// §6.9/§3.10(a') — overlay the pending stall after the common mirror refresh.
METHOD PROTECTED _M_PublishStatus
SUPER^._M_PublishStatus();
// §8.11.4(f)/§8.11.3 — one declaration, two views. Derived AFTER dispatch so the
// wait class reflects the step record this scan just set, not the previous one.
// §3.13 — live row state for the flow chart: how long the active step has run,
// and whether it outran its declared guard (the same watchdog §6.9 stalls on).
IF _exec = E_ExecState.BUSY THEN
    CurrentStepElapsed := DWORD_TO_TIME(TIME_TO_DWORD(TIME()) - _stepSinceMs);
ELSE
    CurrentStepElapsed := T#0S;
END_IF
CurrentStepTimedOut := _tStall.Q;
Starved := (_exec = E_ExecState.BUSY) AND (CurrentStep.TimeClass = E_TimeClass.WAIT_UPSTREAM);
Blocked := (_exec = E_ExecState.BUSY) AND (CurrentStep.TimeClass = E_TimeClass.WAIT_DOWNSTREAM);
// §8.11.3 — classify into the fixed machine-state set (priority: fault first,
// then planned states, then line attribution, then producing/idle).
IF (_exec = E_ExecState.ERROR) OR AlarmLog.Blocking THEN
    MachineState := E_MachineState.DOWN;
ELSIF _mode = E_Mode.CHANGEOVER THEN
    MachineState := E_MachineState.CHANGEOVER;
ELSIF Blocked THEN
    MachineState := E_MachineState.BLOCKED;
ELSIF Starved THEN
    MachineState := E_MachineState.STARVED;
ELSIF _exec = E_ExecState.BUSY THEN
    MachineState := E_MachineState.PRODUCING;
ELSIF _stopReq OR (_exec = E_ExecState.ABORTED) THEN
    MachineState := E_MachineState.STOPPED;
ELSE
    MachineState := E_MachineState.IDLE;
END_IF
Status.ControlDomainId := ControlDomain.Id;
Domain := ControlDomain;
Safety := ControlDomain.Safety;             // read-only HMI mirror; ownership stays in domain
ControlPower := ControlDomain.ControlPower;
IF (_exec <> E_ExecState.ERROR) AND (Pending.ReasonCode <> E_Reason.NONE) THEN
    Status.Diagnostic := Pending;
END_IF
END_METHOD

// §6.9(a) — fixed ring, newest at HistoryHead; never allocates
METHOD PROTECTED _M_PushHistory
VAR_INPUT
    D : ST_Diagnostic;
END_VAR
HistoryHead := (HistoryHead MOD PL_Fraktal.MAX_DIAG_RING) + 1;
History[HistoryHead] := D;
END_METHOD

// §8.11.4(d)/§8.12 — a Low-severity maintenance event: informs planning, does not
// stop the cycle. Instant come+gone ring entry (the trend data lives in Profiler).
METHOD PROTECTED _M_RaiseMaintenance
VAR_INPUT
    Reason : E_Reason;
    Text : STRING(255);
END_VAR
VAR
    slot : INT;
END_VAR
slot := AlarmLog.Raise(Reason := Reason, Text := Text, Source := _name,
    Severity := E_Severity.LOW, Category := E_Category.SYSTEM,
    ResetClass := E_ResetClass.AUTO_RESET);
IF slot > 0 THEN
    AlarmLog.Gone(Slot := slot);
END_IF
END_METHOD

// §3.8b — route a published editable field to the module that registered it.
// WriteConfig already owns access and root-path checks; the recursive walk finds
// the owner by Scope, and that module rechecks revision, type, range, domain and
// its own invariants before storing. A type whose values are declared through
// M_RegisterConfig* therefore needs no override at all, which is the point: a new
// module type costs no routing code (§1.1 O1). Framework-owned keys never reach
// here — _M_WriteBaseConfig answers those first. An override that adds
// hand-written routing shall call SUPER^ first and keep its own answer only when
// the base declines.
METHOD PROTECTED _M_RouteConfigWrite : BOOL
VAR_INPUT
    TargetPath : STRING(255);
    WriteKey   : STRING(160);
    Revision   : UDINT;
    TextValue  : STRING(255);
END_VAR
// RequiresReady is a question about THIS root's state, which the owning child
// cannot see from where it sits, so the root answers it on the way down.
_M_RouteConfigWrite := M_ApplyConfigWrite(Scope := TargetPath,
    WriteKey := WriteKey, Revision := Revision, TextValue := TextValue,
    // Another model's record is not what the machine is running on.
    RootReady := (_exec = E_ExecState.READY) OR (_pModelView <> 0));
END_METHOD

// Framework-owned typed handlers. Stable keys are independent of browse paths;
// capability revision 1 accepts exact enum ordinals and only while READY.
//
// Commit := FALSE validates and stores nothing — the staging pass of a §3.8b set
// load. The root's own ModePolicy keys are published as STATION_CFG
// capabilities, so they are in every station set and have to stage through the
// same validator that writes them, for the same reason every module's do.
METHOD PRIVATE _M_WriteBaseConfig : BOOL
VAR_INPUT
    TargetPath : STRING(255);
    WriteKey   : STRING(160);
    Revision   : UDINT;
    TextValue  : STRING(255);
    Commit     : BOOL;
END_VAR
VAR
    i      : INT;
    key    : STRING(160);
    shield : E_ModeSwitchShield;
    style  : E_ModeSwitchStyle;
END_VAR
_M_WriteBaseConfig := FALSE;
IF (TargetPath <> Status.Name) OR (Revision <> 1) OR (_exec <> E_ExecState.READY) THEN
    RETURN;
END_IF
FOR i := 0 TO PL_Fraktal.MODE_COUNT - 1 DO
    key := CONCAT('unit.modePolicy.', CONCAT(TO_STRING(i), '.shield'));
    IF WriteKey = key THEN
        IF TextValue = '0' THEN
            shield := E_ModeSwitchShield.INTERRUPTIBLE;
        ELSIF TextValue = '1' THEN
            shield := E_ModeSwitchShield.CONFIRM;
        ELSIF TextValue = '2' THEN
            shield := E_ModeSwitchShield.BLOCKED_WHILE_RUNNING;
        ELSE
            RETURN;
        END_IF
        IF Commit THEN
            ModePolicy[i].Shield := shield;
            _modePolicyStored[i].Shield := shield;
        END_IF
        _M_WriteBaseConfig := TRUE;
        RETURN;
    END_IF
    key := CONCAT('unit.modePolicy.', CONCAT(TO_STRING(i), '.style'));
    IF WriteKey = key THEN
        IF TextValue = '0' THEN
            style := E_ModeSwitchStyle.GRACEFUL;
        ELSIF TextValue = '1' THEN
            style := E_ModeSwitchStyle.IMMEDIATE;
        ELSE
            RETURN;
        END_IF
        IF Commit THEN
            ModePolicy[i].Style := style;
            _modePolicyStored[i].Style := style;
        END_IF
        _M_WriteBaseConfig := TRUE;
        RETURN;
    END_IF
END_FOR
END_METHOD

// Application override resolves ChannelPath in THIS root's approved I/O catalog,
// refuses input/safety/unmapped channels, applies its channel-specific §7.6 permit,
// and routes only an approved mapped output. ForceChannel already owns MANUAL,
// stopped/READY, access and audit. Base fails closed.
METHOD PROTECTED _M_RouteForceChannel : BOOL
VAR_INPUT
    ChannelPath : STRING(255);
    Force       : BOOL;
    BoolText    : STRING(255);
    AnalogText  : STRING(160);
END_VAR
_M_RouteForceChannel := FALSE;
END_METHOD

// §7.6.1 — route a manual command to the module that owns TargetPath, through
// the SAME registered-child walk that already carries configuration writes.
//
// This used to return FALSE and leave every Unit to hand-write its own routing
// chain. That is a call a project must remember for correctness (§1.1 O1), and
// it failed exactly as O1 predicts: the press registered eight children and
// routed three, so five modules published manual commands the HMI rendered and
// the Unit silently refused. A registered child is now commandable BECAUSE it
// is registered.
//
// An override still wins, so a Unit with genuinely special routing keeps it;
// it should call SUPER^ first and keep its own answer only when the base
// declines.
METHOD PROTECTED _M_RouteManual : BOOL
VAR_INPUT
    TargetPath : STRING(255);
    Value : DINT;
END_VAR
_M_RouteManual := M_ApplyManual(Scope := TargetPath, Value := Value);
END_METHOD

// §3.13 — keep the published flow chart in step with the chain.
// Called only from _M_SetStep, so every step of every chain lands here exactly
// once per visit and a chain author writes nothing (§1.1 O1). Rows are matched by
// StepNo, appended on first sight and bounded: an overflowing chain publishes the
// first MAX_SEQUENCE_STEPS rows rather than dropping the chart.
METHOD PROTECTED _M_RecordSequenceStep
VAR_INPUT
    StepNo        : INT;
    StepName      : STRING(120);
    Awaits        : I_Module;
    AwaitingLabel : STRING(120);
    TimeClass     : E_TimeClass;
    ExpectedTime  : TIME;
    Branch        : INT;           // §6.12 concurrent leg, 0 = the chain's main line
END_VAR
VAR
    i    : INT;
    hit  : INT;
    path : STRING(255);
END_VAR
hit := 0;
FOR i := 1 TO SequenceStepCount DO
    IF SequenceStepDef[i].StepNo = StepNo THEN
        hit := i;
        EXIT;
    END_IF
END_FOR
IF hit = 0 THEN
    IF SequenceStepCount >= PL_Fraktal.MAX_SEQUENCE_STEPS THEN
        RETURN;                        // bounded: publish what fits, never overrun
    END_IF
    SequenceStepCount := SequenceStepCount + 1;
    hit := SequenceStepCount;
    // §3.10.2 — the static half of this row (StepNo, StepName, the awaited path)
    // is served through the manifest, NOT cyclically, and the HMI refetches only
    // when ConfigRev changes. Rows are discovered by visit, so a chart that grows
    // after the HMI's fetch would render every new row with StepNo 0 and no text.
    // Only the append marks it: a re-visit rewrites identical values.
    //
    // MARKED, not bumped: the revision is raised once the chart stops growing
    // (_M_ChartRevCyclic). Invalidating the whole manifest per discovered row
    // made entering a 15-step mode cost fifteen full refetches.
    _chartDirty := TRUE;
    _chartTouchedMs := TIME_TO_DWORD(TIME());
END_IF
// The drill-down target is the module the step DECLARES it commands. Reading it
// here is what makes the link unambiguous: no IF/CASE chose it (§3.13).
path := '';
IF Awaits <> 0 THEN
    path := Awaits.Name;
END_IF
// Static half: fixed from this first visit, published through the manifest.
SequenceStepDef[hit].StepNo        := StepNo;
SequenceStepDef[hit].Branch        := Branch;
SequenceStepDef[hit].TimeClass     := TimeClass;
SequenceStepDef[hit].ExpectedTime  := ExpectedTime;
SequenceStepDef[hit].StepName      := StepName;
SequenceStepDef[hit].AwaitingLabel := AwaitingLabel;
SequenceStepDef[hit].AwaitsPath    := path;
SequenceSteps[hit].Visited := TRUE;
// §6.12 — the LEG owns the clock, because a leg runs exactly one step at a time.
// A different row on this leg means the step just changed.
IF ActiveSteps[Branch].RowIdx <> hit THEN
    SequenceSteps[hit].WarningActive := FALSE;   // §6.9(e) this visit starts clean
    _M_SequenceAnnotationClear(RowIdx := hit, IsError := FALSE);
    _branchSinceMs[Branch] := TIME_TO_DWORD(TIME());
    ActiveSteps[Branch].RowIdx := hit;
    ActiveSteps[Branch].Elapsed := T#0S;
    ActiveSteps[Branch].TimedOut := FALSE;
    IF Branch = 0 THEN
        _stepSinceMs := _branchSinceMs[0];
        CurrentStepElapsed := T#0S;
    END_IF
END_IF
_branchTouched[Branch] := TRUE;
ActiveSteps[Branch].Elapsed :=
    DWORD_TO_TIME(TIME_TO_DWORD(TIME()) - _branchSinceMs[Branch]);
// A leg carries its own guard: the §6.9 stall watchdog is singular and follows the
// main line, so without this a leg could overrun for ever with nothing to show.
ActiveSteps[Branch].TimedOut := (ExpectedTime > T#0S)
    AND (ActiveSteps[Branch].Elapsed > ExpectedTime);
// The row recorded last IS the step action executing right now, which is what makes
// it the correct target for a §6.9 raise or a §6.9(e) message raised further down
// that same action - on the main line or on any leg.
_seqIndex := hit;
END_METHOD

// §3.13 — drop the published flow chart so the next mode builds its own.
//
// The row table is DISCOVERED by visit (§6.5), which is what makes it free to
// author - but discovery has no end: without this the table becomes the union of
// every chain run since boot. After AUTO then HOME the operator would be shown
// AUTO's rows and HOME's together with only some of them live, and the union of
// the press demo's three modes is 29 rows against a bound of 32. A mode is the
// natural boundary: within one mode a re-run keeps its rows, so Visited and
// LastDuration stay meaningful across cycles.
//
// Bounded by the count actually in use, not by MAX_SEQUENCE_STEPS: clearing rows
// nobody published would cost the whole table on every mode change (§1.1 O10 -
// deterministic scan time).
METHOD PROTECTED _M_ResetSequenceRows
VAR
    i : INT;
    e : ST_SequenceStep;
    x : ST_SequenceStepDef;
    c : ST_SequenceCursor;
    a : ST_SequenceAnnotation;
END_VAR
IF SequenceStepCount > 0 THEN
    // §3.10.2 — the rows this clears are published through the manifest, so the
    // HMI's cached copy is now describing a chart that no longer exists. Guarded
    // by the count: a mode change with nothing published changed no manifest and
    // must not cost a refetch.
    //
    // Marked rather than bumped, and for the same reason as the append: the
    // clear and the regrow that follows it are ONE episode, so they should cost
    // one refetch between them, not one plus one per rediscovered row.
    _chartDirty := TRUE;
    _chartTouchedMs := TIME_TO_DWORD(TIME());
END_IF
FOR i := 1 TO SequenceStepCount DO
    SequenceSteps[i] := e;             // zero-initialized local: clears every field
    SequenceStepDef[i] := x;
END_FOR
SequenceStepCount := 0;
FOR i := 0 TO PL_Fraktal.MAX_PARALLEL_BRANCHES DO
    ActiveSteps[i] := c;
    _branchTouched[i] := FALSE;
END_FOR
FOR i := 1 TO SequenceAnnotationCount DO
    SequenceAnnotations[i] := a;
END_FOR
SequenceAnnotationCount := 0;
_seqIndex := 0;                        // nothing to stamp until the new chain steps
CurrentStepElapsed := T#0S;
END_METHOD

// §6.9 — attach an error or a message to a flow-chart row.
//
// One slot per (row, kind): re-annotating the same row with the same kind
// overwrites rather than accumulating, which is what makes it safe for the
// per-visit message latch to call this without tracking slots.
//
// Returns FALSE when the table is full. The CALLER has already set the row flag
// by then, deliberately: a full table costs the text, never the mark, so the
// chart still shows that something happened here (§5.6 degrade, never mislead).
METHOD PROTECTED _M_SequenceAnnotate : BOOL
VAR_INPUT
    RowIdx     : INT;
    IsError    : BOOL;
    Key        : STRING(120);
    SourcePath : STRING(80);
END_VAR
VAR
    i    : INT;
    slot : INT;
END_VAR
_M_SequenceAnnotate := FALSE;
IF (RowIdx < 1) OR (RowIdx > SequenceStepCount) THEN
    RETURN;
END_IF
slot := 0;
FOR i := 1 TO SequenceAnnotationCount DO
    IF (SequenceAnnotations[i].RowIdx = RowIdx)
    AND (SequenceAnnotations[i].IsError = IsError) THEN
        slot := i;
        EXIT;
    END_IF
END_FOR
IF slot = 0 THEN
    FOR i := 1 TO SequenceAnnotationCount DO
        IF SequenceAnnotations[i].RowIdx = 0 THEN     // freed by a clear
            slot := i;
            EXIT;
        END_IF
    END_FOR
END_IF
IF slot = 0 THEN
    IF SequenceAnnotationCount >= PL_Fraktal.MAX_SEQUENCE_ANNOTATIONS THEN
        RETURN;                                       // full: the mark stands, the text does not
    END_IF
    SequenceAnnotationCount := SequenceAnnotationCount + 1;
    slot := SequenceAnnotationCount;
END_IF
SequenceAnnotations[slot].RowIdx     := RowIdx;
SequenceAnnotations[slot].IsError    := IsError;
SequenceAnnotations[slot].Key        := Key;
SequenceAnnotations[slot].SourcePath := SourcePath;
_M_SequenceAnnotate := TRUE;
END_METHOD

// §6.9 — release annotations. RowIdx 0 means "every row" (the ERROR-cleared edge
// drops all error notes at once); otherwise just that row's note of that kind.
// Freed slots are reused before the table grows, so a chain that warns on many
// steps over many cycles does not exhaust it.
METHOD PROTECTED _M_SequenceAnnotationClear
VAR_INPUT
    RowIdx  : INT;
    IsError : BOOL;
END_VAR
VAR
    i : INT;
    e : ST_SequenceAnnotation;
END_VAR
FOR i := 1 TO SequenceAnnotationCount DO
    IF (SequenceAnnotations[i].IsError = IsError)
    AND ((RowIdx = 0) OR (SequenceAnnotations[i].RowIdx = RowIdx)) THEN
        SequenceAnnotations[i] := e;                  // RowIdx 0 marks the slot free
    END_IF
END_FOR
END_METHOD

// §6.5 — the ONE line per step: record for the §6.9 walk AND the §8.11.4 profiler
METHOD PROTECTED _M_SetStep
VAR_INPUT
    StepNo        : INT;
    StepName      : STRING(120);
    Awaits        : I_Module;
    AwaitingLabel : STRING(120);
    TimeClass     : E_TimeClass;
    ExpectedTime  : TIME;
END_VAR
VAR
    i : INT;
    e : ST_CondRecord;
END_VAR
IF StepNo <> CurrentStep.StepNo THEN
    _tStall(IN := FALSE);
    _M_ClearPending();
    FOR i := 1 TO PL_Fraktal.MAX_STEP_CONDS DO
        CurrentStep.Conds[i] := e;
    END_FOR
END_IF
CurrentStep.StepNo        := StepNo;
CurrentStep.StepName      := StepName;
CurrentStep.AwaitingLabel := AwaitingLabel;
CurrentStep.TimeClass     := TimeClass;
CurrentStep.ExpectedTime  := ExpectedTime;
_awaits := Awaits;
_M_RecordSequenceStep(StepNo := StepNo, StepName := StepName, Awaits := Awaits,
    AwaitingLabel := AwaitingLabel, TimeClass := TimeClass, ExpectedTime := ExpectedTime,
    Branch := 0);
Profiler.StepChanged(StepNo := StepNo, StepName := StepName, TimeClass := TimeClass,
    Expected := ExpectedTime);
END_METHOD

// §6.9 — build the pending stall reason: step -> awaited command -> first FALSE condition
METHOD PROTECTED _M_StallWalk
IF Pending.ReasonCode = E_Reason.NONE THEN
    Pending.Since := F_Now();
    Pending.TimeSynchronized := F_TimeSynchronized();
END_IF
Pending.ReasonCode := E_Reason.STEP_STALLED;
Pending.Severity   := E_Severity.LOW;
Pending.Category   := E_Category.PROCESS;
Pending.SourcePath := _name;
Pending.Description := 'std.diagnostic.stepStalled';
END_METHOD

// §3.4.2 — the sequence author calls this at each step boundary; returns TRUE when
// the sequence may advance. Steppable (default TRUE) is the PER-STEP stop-point flag:
// a step with Steppable := FALSE runs straight through even in SINGLE_STEP/HOLD_TO_RUN
// (group several motions into one operator step, or a step unsafe to pause mid-way).
// CONTINUOUS: always TRUE. SINGLE_STEP: TRUE once per StepRequest edge (only if
// Steppable). HOLD_TO_RUN: TRUE while held (only if Steppable). Interlocks are
// enforced by the modules regardless (this only paces the sequence).
METHOD PROTECTED _M_StepGate : BOOL
VAR_INPUT
    Steppable : BOOL;
END_VAR
IF NOT Steppable THEN
    _M_StepGate := TRUE;               // not a stop point: advance regardless of run style
    RETURN;
END_IF
CASE RunStyle OF
    E_RunStyle.SINGLE_STEP:
        _stepArm(CLK := _stepReq);
        _stepReq := FALSE;
        _M_StepGate := _stepArm.Q;      // one advance per request edge
    E_RunStyle.HOLD_TO_RUN:
        _M_StepGate := _holdRun;        // advance only while held (NON-SAFETY)
ELSE
    _M_StepGate := TRUE;                // CONTINUOUS
END_CASE
END_METHOD

// §3.4 — override to declare the type's mode set (baseline: AUTO + MANUAL)
METHOD PROTECTED _M_Supports : BOOL
VAR_INPUT
    Mode : E_Mode;
END_VAR
_M_Supports := (Mode = E_Mode.AUTO) OR (Mode = E_Mode.MANUAL);
END_METHOD

// §3.4.2 — a concrete Unit overrides to opt a mode into SINGLE_STEP/HOLD_TO_RUN.
// Base: only CONTINUOUS.
METHOD PROTECTED _M_SupportsRunStyle : BOOL
VAR_INPUT
    Style : E_RunStyle;
END_VAR
_M_SupportsRunStyle := (Style = E_RunStyle.CONTINUOUS);
END_METHOD

// §6.11 — returns the chosen option once and clears the request (0 = none yet)
METHOD PROTECTED _M_TakeDecision : INT
IF DecisionAnswer > 0 THEN
    _M_TakeDecision := DecisionAnswer;
    IF NOT _decisionResolutionLogged THEN
        _M_LogDecision(EventKey := 'std.audit.decisionOperatorResolved',
            SourcePath := Decision.SourcePath, Option := DecisionAnswer);
    END_IF
    _M_ClearDecisionState();
ELSE
    _M_TakeDecision := 0;
END_IF
END_METHOD

// §8.11 — called by the chain/verdict glue at part completion
METHOD CountGood : BOOL
GoodCount := GoodCount + 1;
CountGood := TRUE;
END_METHOD

// Sections 8.11.2 and 11.6: one authoritative NOK outcome path.
// Part.Uid is empty when the optional traceability carrier is not configured.
METHOD CountNok : BOOL
VAR_INPUT
    Reason : E_Reason;
END_VAR
CountNok := FALSE;
IF Reason = E_Reason.NONE THEN
    _M_Fault(E_Reason.RESULT_RECORD_REJECTED, 'std.error.nokReasonRequired');
    RETURN;
END_IF
IF NOT _M_HostEvent(Kind := E_HostEventKind.NOK, PartUid := Part.Uid,
        Subject := '', Value := '', Verdict := E_Verdict.NOK,
        ReasonCode := Reason) THEN
    _M_Fault(E_Reason.RESULT_RECORD_REJECTED, 'std.error.hostEventRejected');
    RETURN;
END_IF
NokCount := NokCount + 1;
NokReason := Reason;
CountNok := TRUE;
END_METHOD

// §8.11.2 — REWORK verdict counter (see CountGood)
METHOD CountRework : BOOL
ReworkCount := ReworkCount + 1;
CountRework := TRUE;
END_METHOD

// §3.10.2 — Unit facets after the composite walk (own catalog + children):
// model catalog and per-mode switch policy, both static between config edits.
METHOD M_AppendConfig : BOOL
VAR_INPUT
    Pager : REFERENCE TO FB_ConfigPager;
END_VAR
VAR
    i        : INT;
    metaIndex: INT;
    item     : STRING(255);
    writeKey : STRING(160);
    labelKey : STRING(160);  // std.config.modePolicy.<mode ordinal>.<shield|style>
    meta     : ST_AlarmMeta;
    seqIdx   : INT;
    seqBase  : STRING(255);
END_VAR
M_AppendConfig := SUPER^.M_AppendConfig(Pager := Pager);
IF _pLine <> 0 THEN
    _pLine^.M_AppendLineConfig(Pager := Pager, Scope := Status.Name);   // §3.8e
END_IF
Pager.M_AppendNumber(Scope := Status.Name, Item := 'StallTime',
    Number := TIME_TO_DINT(StallTime));
Pager.M_Append(Scope := Status.Name, Item := 'ModelCapacity',
    ValueText := TO_STRING(ModelCapacity));
Pager.M_Append(Scope := Status.Name, Item := 'Features/ExportCurrentConfig',
    ValueText := TO_STRING(Features.ExportCurrentConfig));
Pager.M_AppendNumber(Scope := Status.Name, Item := 'AvailableModelCount',
    Number := TO_DINT(AvailableModelCount));
FOR i := 1 TO AvailableModelCount DO
    item := CONCAT('AvailableModels/AvailableModels[',
        CONCAT(TO_STRING(i), ']/ModelCode'));
    Pager.M_Append(Scope := Status.Name, Item := item,
        ValueText := AvailableModels[i].ModelCode);
END_FOR
FOR i := 0 TO PL_Fraktal.MODE_COUNT - 1 DO
    item := CONCAT('ModePolicy/ModePolicy[', CONCAT(TO_STRING(i), ']/Shield'));
    writeKey := CONCAT('unit.modePolicy.', CONCAT(TO_STRING(i), '.shield'));
    labelKey := CONCAT('std.config.modePolicy.', CONCAT(TO_STRING(i), '.shield'));
    Pager.M_AppendCapability(Scope := Status.Name, Item := item,
        ValueText := TO_STRING(TO_DINT(ModePolicy[i].Shield)), WriteKey := writeKey,
        WriteRevision := 1, ConfigKind := E_ConfigKind.STATION_CFG,
        ValueType := E_ConfigValueType.NUMBER, Writable := TRUE,
        RequiresReady := TRUE, HasMinimum := TRUE, HasMaximum := TRUE,
        Minimum := 0.0, Maximum := 2.0, Unit := E_EngUnit.NONE, LabelKey := labelKey,
        EnumDomain := '0|1|2', EnumLabelKey := 'std.enum.modeSwitchShield',
        ClassId := '', MinReadLevel := E_AccessLevel.NONE,
        MinWriteLevel := E_AccessLevel.NONE, ModelScoped := FALSE);
    item := CONCAT('ModePolicy/ModePolicy[', CONCAT(TO_STRING(i), ']/Style'));
    writeKey := CONCAT('unit.modePolicy.', CONCAT(TO_STRING(i), '.style'));
    labelKey := CONCAT('std.config.modePolicy.', CONCAT(TO_STRING(i), '.style'));
    Pager.M_AppendCapability(Scope := Status.Name, Item := item,
        ValueText := TO_STRING(TO_DINT(ModePolicy[i].Style)), WriteKey := writeKey,
        WriteRevision := 1, ConfigKind := E_ConfigKind.STATION_CFG,
        ValueType := E_ConfigValueType.NUMBER, Writable := TRUE,
        RequiresReady := TRUE, HasMinimum := TRUE, HasMaximum := TRUE,
        Minimum := 0.0, Maximum := 1.0, Unit := E_EngUnit.NONE, LabelKey := labelKey,
        EnumDomain := '0|1', EnumLabelKey := 'std.enum.modeSwitchStyle',
        ClassId := '', MinReadLevel := E_AccessLevel.NONE,
        MinWriteLevel := E_AccessLevel.NONE, ModelScoped := FALSE);
END_FOR
Pager.M_AppendNumber(Scope := Status.Name, Item := 'AlarmLog/MetaCount',
    Number := TO_DINT(PL_ReasonCatalog.COUNT + AlarmLog.MetaCount));
// §8.8/§8.9: the standard catalog is generated from the numeric sources plus
// one symbol-keyed rationalization registry. Static metadata stays manifest-only.
FOR i := 1 TO PL_ReasonCatalog.COUNT DO
    IF NOT F_ReasonMetaByIndex(Index := i, Meta := meta) THEN
        EXIT;
    END_IF
    item := CONCAT('AlarmLog/Meta/Meta[', CONCAT(TO_STRING(i), ']/ReasonCode'));
    Pager.M_AppendNumber(Scope := Status.Name, Item := item,
        Number := TO_DINT(meta.ReasonCode));
    item := CONCAT('AlarmLog/Meta/Meta[', CONCAT(TO_STRING(i), ']/OperatorAction'));
    Pager.M_Append(Scope := Status.Name, Item := item,
        ValueText := meta.OperatorAction);
    item := CONCAT('AlarmLog/Meta/Meta[', CONCAT(TO_STRING(i), ']/Consequence'));
    Pager.M_Append(Scope := Status.Name, Item := item,
        ValueText := meta.Consequence);
    item := CONCAT('AlarmLog/Meta/Meta[', CONCAT(TO_STRING(i), ']/Priority'));
    Pager.M_AppendNumber(Scope := Status.Name, Item := item,
        Number := TO_DINT(meta.Priority));
    item := CONCAT('AlarmLog/Meta/Meta[', CONCAT(TO_STRING(i), ']/Category'));
    Pager.M_AppendNumber(Scope := Status.Name, Item := item,
        Number := TO_DINT(meta.Category));
    item := CONCAT('AlarmLog/Meta/Meta[', CONCAT(TO_STRING(i), ']/Shelvable'));
    IF meta.Shelvable THEN
        Pager.M_Append(Scope := Status.Name, Item := item, ValueText := 'TRUE');
    ELSE
        Pager.M_Append(Scope := Status.Name, Item := item, ValueText := 'FALSE');
    END_IF
END_FOR
// External/application libraries may append rationalized reasons not present in
// the shipped registry. RegisterMetaFull enforces their complete record.
FOR i := 1 TO AlarmLog.MetaCount DO
    metaIndex := PL_ReasonCatalog.COUNT + i;
    item := CONCAT('AlarmLog/Meta/Meta[', CONCAT(TO_STRING(metaIndex), ']/ReasonCode'));
    Pager.M_AppendNumber(Scope := Status.Name, Item := item,
        Number := TO_DINT(AlarmLog.Meta[i].ReasonCode));
    item := CONCAT('AlarmLog/Meta/Meta[', CONCAT(TO_STRING(metaIndex), ']/OperatorAction'));
    Pager.M_Append(Scope := Status.Name, Item := item,
        ValueText := AlarmLog.Meta[i].OperatorAction);
    item := CONCAT('AlarmLog/Meta/Meta[', CONCAT(TO_STRING(metaIndex), ']/Consequence'));
    Pager.M_Append(Scope := Status.Name, Item := item,
        ValueText := AlarmLog.Meta[i].Consequence);
    item := CONCAT('AlarmLog/Meta/Meta[', CONCAT(TO_STRING(metaIndex), ']/Priority'));
    Pager.M_AppendNumber(Scope := Status.Name, Item := item,
        Number := TO_DINT(AlarmLog.Meta[i].Priority));
    item := CONCAT('AlarmLog/Meta/Meta[', CONCAT(TO_STRING(metaIndex), ']/Category'));
    Pager.M_AppendNumber(Scope := Status.Name, Item := item,
        Number := TO_DINT(AlarmLog.Meta[i].Category));
    item := CONCAT('AlarmLog/Meta/Meta[', CONCAT(TO_STRING(metaIndex), ']/Shelvable'));
    IF AlarmLog.Meta[i].Shelvable THEN
        Pager.M_Append(Scope := Status.Name, Item := item, ValueText := 'TRUE');
    ELSE
        Pager.M_Append(Scope := Status.Name, Item := item, ValueText := 'FALSE');
    END_IF
END_FOR
// §3.13/§3.10.2 — the static definition of each flow-chart row. The Item fragment
// reproduces the browse path the LIVE half is published under, so the HMI mapper
// reads `SequenceSteps[i]/StepName` without knowing it arrived by a different
// route: one row structure, half of it live, half fetched once and cached.
// Bounded by the discovered count, so an empty chain appends nothing.
FOR seqIdx := 1 TO SequenceStepCount DO
    seqBase := CONCAT('SequenceSteps/SequenceSteps[', CONCAT(TO_STRING(seqIdx), ']/'));
    Pager.M_AppendNumber(Scope := Status.Name, Item := CONCAT(seqBase, 'StepNo'),
        Number := TO_DINT(SequenceStepDef[seqIdx].StepNo));
    Pager.M_AppendNumber(Scope := Status.Name, Item := CONCAT(seqBase, 'Branch'),
        Number := TO_DINT(SequenceStepDef[seqIdx].Branch));
    Pager.M_AppendNumber(Scope := Status.Name, Item := CONCAT(seqBase, 'TimeClass'),
        Number := TO_DINT(SequenceStepDef[seqIdx].TimeClass));
    Pager.M_AppendNumber(Scope := Status.Name, Item := CONCAT(seqBase, 'ExpectedTime'),
        Number := TIME_TO_DINT(SequenceStepDef[seqIdx].ExpectedTime));
    Pager.M_Append(Scope := Status.Name, Item := CONCAT(seqBase, 'StepName'),
        ValueText := SequenceStepDef[seqIdx].StepName);
    Pager.M_Append(Scope := Status.Name, Item := CONCAT(seqBase, 'AwaitingLabel'),
        ValueText := SequenceStepDef[seqIdx].AwaitingLabel);
    Pager.M_Append(Scope := Status.Name, Item := CONCAT(seqBase, 'AwaitsPath'),
        ValueText := SequenceStepDef[seqIdx].AwaitsPath);
END_FOR
END_METHOD

// §3.8b — inject this deployment's parameter-set store at Setup, the same shape
// as SetPartCarrier and the §3.8 recipe provider. Absent means save/load/list are
// not offered at all, published as StorePresent = FALSE — a stated fact rather
// than a request that fails the first time an operator tries it.
METHOD SetConfigStore : BOOL
VAR_INPUT
    Store : I_ConfigStore;
END_VAR
SetConfigStore := FALSE;
IF Store = 0 THEN
    RETURN;
END_IF
_configStore := Store;
// A store that writes its own sets out is a durability provider as well.
IF NOT __QUERYINTERFACE(Store, _storePersistence) THEN
    _storePersistence := 0;
END_IF
ConfigPersist.StorePresent := TRUE;
ConfigPersist.StoreKind := Store.M_Kind();
SetConfigStore := TRUE;
END_METHOD

// §3.8b - keep this root's live configuration on the project's medium too: the
// station data, the line data this root owns, and every model's data, one
// document each ('<root>.station', '<root>.line', '<root>.model<n>'). At start
// the documents are read back and replayed through the owning handlers, staged
// and all-or-nothing per document, before any configuration write is accepted;
// after every accepted write they are written again. A missing document is a
// first start. One the medium confirmed and then lost, or one that no longer
// fits this build, is announced as a lost image under its key (§3.8b restore).
// The native PERSISTENT data stays: it seeds the first documents and is what a
// lost one falls back to. The same medium may serve the set store and the
// access provider. Refused once the restore has started.
METHOD SetPersistMedium : BOOL
VAR_INPUT
    Medium : I_PersistMedium;
END_VAR
SetPersistMedium := FALSE;
IF (Medium = 0) OR (_livePhase <> 0) THEN
    RETURN;
END_IF
_medium := Medium;
SetPersistMedium := TRUE;
END_METHOD

// §3.8b — substitute the durability provider. The shipped LOCAL_RETAIN writer is
// used when nothing is injected, so this exists for a deployment whose
// configuration genuinely lives somewhere else (a file, a database, an MES) —
// not as one more thing every station has to remember to wire (§1.1 O1).
METHOD SetConfigPersistence : BOOL
VAR_INPUT
    Provider : I_ConfigPersistence;
END_VAR
SetConfigPersistence := FALSE;
IF Provider = 0 THEN
    RETURN;
END_IF
_persistence := Provider;
SetConfigPersistence := TRUE;
END_METHOD

// §3.8b — declare how long an accepted write may take to become durable. The
// clause says "within a declared bounded window", and the point of DECLARING it
// is that different stores have honestly different latencies: a retentive write
// is milliseconds, an MES round trip is not. A deployment that leaves this alone
// gets PL_Fraktal.CONFIG_PERSIST_WINDOW_MS.
//
// Zero means "durable immediately or not at all", which is the correct
// declaration for a store that either completes in the same scan or has failed.
METHOD SetConfigPersistWindow : BOOL
VAR_INPUT
    WindowMs : UDINT;
END_VAR
ConfigPersist.WindowMs := WindowMs;
SetConfigPersistWindow := TRUE;
END_METHOD

// §3.8b — declare what this station DOES about a lost configuration image.
// DEFAULTS_AND_ANNUNCIATE is the shipped default; a station whose commissioned
// values are the difference between a good part and a wrecked tool declares
// BLOCK_UNTIL_ACKNOWLEDGED instead. It is a DEPLOYMENT decision on purpose: no
// module type is in a position to know which of the two its station is, which is
// why a module reporting a loss never decides the consequence of one.
METHOD SetConfigRestorePolicy : BOOL
VAR_INPUT
    Policy : E_ConfigRestorePolicy;
END_VAR
ConfigPersist.RestorePolicy := Policy;
SetConfigRestorePolicy := TRUE;
END_METHOD

// §3.8b — an accepted write is LIVE. This starts the clock on it becoming
// DURABLE, and the root publishes PersistPending until it is. Called from every
// path that accepts a value, so no project and no module type has to remember
// that a write it just made is not yet safe (§1.1 O1).
METHOD PROTECTED _M_MarkPersistPending
IF NOT ConfigPersist.Pending THEN
    ConfigPersist.Pending := TRUE;
    ConfigPersist.PendingSince := F_Now();
END_IF
// The window runs from the LATEST accepted write, because that is the one whose
// durability is in question; PendingSince stays at the start of the episode so
// an operator can see how long this station has been unsafe.
_persistSinceMs := TIME_TO_DWORD(TIME());
ConfigPersist.Failed := FALSE;
IF _persistEvt > 0 THEN
    AlarmLog.Gone(Slot := _persistEvt);
    _persistEvt := 0;
END_IF
IF _medium <> 0 THEN
    _liveDirty := TRUE;                    // the live documents follow
    _liveFailed := FALSE;                  // a new write re-arms a failed pass at once
END_IF
IF _storePersistence <> 0 THEN
    IF NOT _storePersistence.M_Request() THEN
        _M_ConfigPersistFailed();
    END_IF
END_IF
IF _persistence = 0 THEN
    RETURN;                                // no provider: the window will expire
END_IF
IF NOT _persistence.M_Request() THEN
    _M_ConfigPersistFailed();              // refused before it began is a failure
END_IF
END_METHOD

// §3.8b — the store rejected the write, or the declared window elapsed with it
// still not durable. Pending stays TRUE because the value is STILL not durable;
// Failed says it will not get there on its own.
//
// Deliberately NOT retried in a loop: a store that cannot write is not fixed by
// asking again every scan, and a retry storm would bury the one annunciation an
// operator needs. The next accepted write re-arms it.
METHOD PRIVATE _M_ConfigPersistFailed
ConfigPersist.Failed := TRUE;
IF _persistEvt > 0 THEN
    RETURN;                                // one standing event, not one per scan
END_IF
// AUTO_RESET: loud enough to see, never blocking. A station whose configuration
// will not persist can still finish the parts already in it, and the operator is
// told BEFORE the restart that would otherwise reveal this silently.
_persistEvt := AlarmLog.Raise(Reason := E_Reason.CONFIG_PERSIST_FAILED,
    Text := 'std.error.configPersistFailed', Source := _name,
    Severity := E_Severity.MED, Category := E_Category.SYSTEM,
    ResetClass := E_ResetClass.AUTO_RESET);
END_METHOD

// §3.8b — drive the durability provider and hold the declared window to
// account. "Within a declared bounded window" is a promise, and a promise
// nobody measures is the hope the clause replaces: the window is checked here
// every scan, and exceeding it publishes PersistFailed.
METHOD PRIVATE _M_ConfigPersistCyclic
VAR
    busy    : BOOL;
    elapsed : DWORD;
END_VAR
busy := FALSE;
IF _persistence <> 0 THEN
    busy := _persistence.M_Cyclic();
END_IF
// A store that writes its sets out, and the live documents, are durability
// providers too: Pending holds until every one of them is done.
IF _storePersistence <> 0 THEN
    IF _storePersistence.M_Cyclic() THEN
        busy := TRUE;
    END_IF
END_IF
IF _M_LiveCyclic() THEN
    busy := TRUE;
END_IF
IF NOT ConfigPersist.Pending THEN
    RETURN;
END_IF
IF busy THEN
    // Unsigned subtraction, so the monotonic millisecond counter wrapping does
    // not fabricate an expired window (TC3 §8.11).
    elapsed := TIME_TO_DWORD(TIME()) - _persistSinceMs;
    IF elapsed > TO_DWORD(ConfigPersist.WindowMs) THEN
        _M_ConfigPersistFailed();
    END_IF
    RETURN;
END_IF
// Nothing in flight. Either it finished, or there is no provider to finish it.
IF _persistence = 0 THEN
    elapsed := TIME_TO_DWORD(TIME()) - _persistSinceMs;
    IF elapsed > TO_DWORD(ConfigPersist.WindowMs) THEN
        _M_ConfigPersistFailed();
    END_IF
    RETURN;
END_IF
IF _persistence.M_Failed() THEN
    _M_ConfigPersistFailed();
    RETURN;
END_IF
IF _liveFailed THEN
    _M_ConfigPersistFailed();
    RETURN;
END_IF
IF _storePersistence <> 0 THEN
    IF _storePersistence.M_Failed() THEN
        _M_ConfigPersistFailed();
        RETURN;
    END_IF
END_IF
ConfigPersist.Pending := FALSE;
ConfigPersist.Failed := FALSE;
IF _persistEvt > 0 THEN
    AlarmLog.Gone(Slot := _persistEvt);
    _persistEvt := 0;
END_IF
END_METHOD

// §3.8b - TRUE once the live documents are back (or there is no medium). Until
// then a configuration write is refused: the restore would replay over it.
METHOD PRIVATE _M_ConfigRestored : BOOL
_M_ConfigRestored := (_medium = 0) OR _liveRestored;
END_METHOD

// §3.8b - read the live documents back once, then write all of them again after
// every accepted change: station, line, then each model. TRUE while a document
// is not yet where it belongs, which holds PersistPending for that long.
//
// One pass rewrites every document rather than tracking which value changed:
// a pass is bounded (2 + MAX_RECIPES documents), and a document written whole
// from the capability walk can never disagree with the machine.
METHOD PRIVATE _M_LiveCyclic : BOOL
VAR
    n          : INT;
    kind       : E_ConfigKind;
    modelIndex : UDINT;
    started    : BOOL;
    refused    : BOOL;     // the medium's queue was full: ask again next scan
END_VAR
_M_LiveCyclic := FALSE;
IF _medium = 0 THEN
    RETURN;
END_IF
CASE _livePhase OF
    0:      // the capability walk is complete once OnInit ran
        IF _liveArmed THEN
            _liveModels := _M_LiveModelsKept();
            _liveItem := 1;
            _livePhase := 10;
        END_IF
    10:     // restore: the next document
        IF _liveItem > 2 + PL_Fraktal.MAX_RECIPES THEN
            _liveRestored := TRUE;
            _livePhase := 30;
            ConfigRev := ConfigRev + 1;    // restored values: the manifest reads differently
            _M_MarkPersistPending();       // every store, and the documents as the new baseline
        ELSIF NOT _M_LiveItemUsed(Item := _liveItem, Restoring := TRUE) THEN
            _liveItem := _liveItem + 1;
        ELSIF _liveDoc.M_Read(Medium := _medium, Key := _M_LiveKey(Item := _liveItem)) THEN
            _livePhase := 11;
        END_IF
    11:
        IF _liveDoc.M_Poll() THEN
            IF _liveDoc.Ok THEN
                _M_LiveRestoreItem();
                _liveItem := _liveItem + 1;
                _livePhase := 10;
            ELSE
                // The medium could not answer: that is not "nothing there". Restoring
                // anyway would run on defaults and write them over the documents.
                _M_LiveReadFailed();
                _liveRetry(IN := FALSE, PT := LIVE_READ_RETRY);
                _livePhase := 12;
            END_IF
        END_IF
    12:     // the same document again after LIVE_READ_RETRY
        _liveRetry(IN := TRUE, PT := LIVE_READ_RETRY);
        IF _liveRetry.Q THEN
            _liveRetry(IN := FALSE, PT := LIVE_READ_RETRY);
            _livePhase := 10;
        END_IF
    30:     // idle: one pass after an accepted change; a failed pass is retried
        _liveRetry(IN := _liveFailed AND _liveDirty, PT := LIVE_RETRY);
        IF _liveDirty AND (NOT _liveFailed OR _liveRetry.Q) THEN
            _liveRetry(IN := FALSE, PT := LIVE_RETRY);
            _liveDirty := FALSE;           // a change during the pass marks it again
            _liveItem := 1;
            _livePhase := 40;
        END_IF
    40:
        IF _liveItem > 2 + PL_Fraktal.MAX_RECIPES THEN
            _liveFailed := FALSE;
            IF _liveModels THEN
                _liveModelSlots := AvailableModelCount;
            END_IF
            _livePhase := 30;
        ELSIF NOT _M_LiveItemUsed(Item := _liveItem, Restoring := FALSE) THEN
            _liveItem := _liveItem + 1;
        ELSE
            n := _liveItem - 2;
            started := FALSE;
            refused := FALSE;
            IF n > AvailableModelCount THEN
                // A model document past the catalog: the model is no longer offered.
                started := _liveDoc.M_Delete(Medium := _medium, Key := _M_LiveKey(Item := _liveItem));
                refused := NOT started AND (_liveDoc.ErrorId = 16#706);
            ELSE
                kind := E_ConfigKind.STATION_CFG;
                modelIndex := 0;
                IF _liveItem = 2 THEN
                    kind := E_ConfigKind.LINE_CFG;
                ELSIF _liveItem > 2 THEN
                    kind := E_ConfigKind.PAR_CFG;
                    modelIndex := INT_TO_UDINT(n);
                END_IF
                IF _M_CaptureInto(Store := _loadSnapshot, SetName := '_live', Kind := kind,
                        ModelIndex := modelIndex) THEN
                    started := _liveDoc.M_Write(Medium := _medium,
                        Key := _M_LiveKey(Item := _liveItem), Store := _loadSnapshot,
                        SetName := '_live');
                    refused := NOT started AND (_liveDoc.ErrorId = 16#706);
                END_IF
            END_IF
            IF started THEN
                _livePhase := 41;
            ELSIF NOT refused THEN
                _M_LivePassFailed();            // not rendered, or the walk did not fit a set
            END_IF
        END_IF
    41:
        IF _liveDoc.M_Poll() THEN
            IF _liveDoc.Ok THEN
                _liveItem := _liveItem + 1;
                _livePhase := 40;
            ELSE
                _M_LivePassFailed();
            END_IF
        END_IF
ELSE
    _livePhase := 30;
END_CASE
_M_LiveCyclic := NOT _liveRestored OR _liveDirty OR (_livePhase = 40) OR (_livePhase = 41);
END_METHOD

// §3.8b - a live document could not be read at start. Announced once (AUTO_RESET,
// gone when the restore completes, through _M_MarkPersistPending); Start meanwhile
// names the restore and configuration writes are refused.
METHOD PRIVATE _M_LiveReadFailed
ConfigPersist.Failed := TRUE;
IF _persistEvt > 0 THEN
    RETURN;
END_IF
_persistEvt := AlarmLog.Raise(Reason := E_Reason.CONFIG_PERSIST_FAILED,
    Text := 'std.error.storageUnreadable', Source := _M_LiveKey(Item := _liveItem),
    Severity := E_Severity.MED, Category := E_Category.SYSTEM,
    ResetClass := E_ResetClass.AUTO_RESET);
END_METHOD

METHOD PRIVATE _M_LivePassFailed
_liveFailed := TRUE;
_liveDirty := TRUE;            // retried after LIVE_RETRY, or at the next write
_livePhase := 30;
END_METHOD

// Which documents this root keeps: always the station; the line only when this
// root hosts a line it owns (a mirror's values are its owner's); a model when
// model data is kept, every slot on restore and, when writing, every model the
// catalog offers plus any older slot still to be cleared.
METHOD PRIVATE _M_LiveItemUsed : BOOL
VAR_INPUT
    Item      : INT;
    Restoring : BOOL;
END_VAR
_M_LiveItemUsed := FALSE;
IF Item = 1 THEN
    _M_LiveItemUsed := TRUE;
ELSIF Item = 2 THEN
    IF (_pLine <> 0) AND _lineHost THEN
        _M_LiveItemUsed := _pLine^.OutImm.Role = E_LineRole.OWNER;
    END_IF
ELSIF _liveModels THEN
    _M_LiveItemUsed := Restoring OR ((Item - 2) <= MAX(AvailableModelCount, _liveModelSlots));
END_IF
END_METHOD

METHOD PRIVATE _M_LiveKey : STRING(80)
VAR_INPUT
    Item : INT;
END_VAR
IF Item = 1 THEN
    _M_LiveKey := CONCAT(Status.Name, '.station');
ELSIF Item = 2 THEN
    _M_LiveKey := CONCAT(Status.Name, '.line');
ELSE
    _M_LiveKey := CONCAT(Status.Name, CONCAT('.model', INT_TO_STRING(Item - 2)));
END_IF
END_METHOD

// Model data is kept per model when this root registered its own record
// (M_RegisterModelData) with a provider that stores records, and every PAR_CFG
// value of the walk lives in that record. A child's model data belongs to the
// child's recipe, which this root cannot select per model.
METHOD PRIVATE _M_LiveModelsKept : BOOL
VAR
    store  : I_RecipeStore;
    info   : ST_ConfigSetInfo;
    record : ST_ConfigRecord;
    i      : INT;
END_VAR
_M_LiveModelsKept := FALSE;
IF (_modelProvider = 0) OR (_pModelRegion = 0) THEN
    RETURN;
END_IF
IF NOT __QUERYINTERFACE(_modelProvider, store) THEN
    RETURN;
END_IF
IF NOT _M_CaptureInto(Store := _loadSnapshot, SetName := '_live',
        Kind := E_ConfigKind.PAR_CFG, ModelIndex := 0) THEN
    RETURN;
END_IF
IF NOT _loadSnapshot.M_ReadInfo(SetName := '_live', Info := info) THEN
    RETURN;
END_IF
FOR i := 1 TO info.RecordCount DO
    IF NOT _loadSnapshot.M_ReadRecord(SetName := '_live', Index := i, Record := record) THEN
        RETURN;
    END_IF
    IF NOT _M_OwnsModelRecord(Record := record) THEN
        RETURN;
    END_IF
END_FOR
_M_LiveModelsKept := TRUE;
END_METHOD

// §3.8b - the medium answered for one document: replay it, or announce why not.
// Nothing there is a first start; nothing there where the medium confirmed a
// write, a document that does not parse or no longer fits this build, or an older
// copy than the one confirmed, is a lost image announced under the document's
// key. The values then stay as they are - the native retained data - and the next
// pass writes them as the new baseline, so the loss is announced once. (A medium
// that could not answer never gets here: _M_LiveCyclic asks again.)
METHOD PRIVATE _M_LiveRestoreItem
VAR
    info     : ST_ConfigSetInfo;
    key      : STRING(80);
    expected : E_ConfigKind;
    applied  : BOOL;
END_VAR
key := _M_LiveKey(Item := _liveItem);
IF NOT _liveDoc.Found THEN
    IF _liveDoc.Lost THEN
        _M_AnnounceRestoreLoss(Path := key, Text := 'std.error.configRestoreLost');
    END_IF
    RETURN;
END_IF
expected := E_ConfigKind.STATION_CFG;
IF _liveItem = 2 THEN
    expected := E_ConfigKind.LINE_CFG;
ELSIF _liveItem > 2 THEN
    expected := E_ConfigKind.PAR_CFG;
    _liveModelSlots := MAX(_liveModelSlots, _liveItem - 2);
END_IF
applied := FALSE;
IF _liveDoc.M_Parse(Store := _loadSnapshot, Info := info) THEN
    IF (info.Kind = expected) AND (info.RootIdentity = Status.Name) THEN
        applied := _M_LiveApply(Info := info);
    END_IF
END_IF
IF NOT applied OR _liveDoc.Lost THEN
    _M_AnnounceRestoreLoss(Path := key, Text := 'std.error.configRestoreLost');
END_IF
END_METHOD

// Replay a restored document frozen in _loadSnapshot through the same staged,
// all-or-nothing path a set load takes. A model document goes into that model's
// record (the live one for the active model) and back to the provider; a model
// created at run time whose catalog record did not survive is created again
// from the live record first, then given its values.
METHOD PRIVATE _M_LiveApply : BOOL
VAR_INPUT
    Info : ST_ConfigSetInfo;
END_VAR
VAR
    index : UDINT;
END_VAR
_M_LiveApply := FALSE;
index := 0;
IF Info.Kind = E_ConfigKind.PAR_CFG THEN
    index := _M_ModelIndexOf(ModelCode := Info.ModelCode);
    IF (index = 0) AND (_modelCatalog <> 0) AND (Info.ModelCode <> '')
    AND (AvailableModelCount < ModelCapacity) THEN
        MEMCPY(destAddr := ADR(_modelBuf), srcAddr := _pModelRegion, n := _modelRegionSize);
        IF _modelCatalog.M_CreateModel(ModelCode := Info.ModelCode, RecipeKey := _modelKey,
                pData := ADR(_modelBuf), Size := _modelRegionSize) THEN
            _M_SyncModelCatalog();
            index := _M_ModelIndexOf(ModelCode := Info.ModelCode);
        END_IF
    END_IF
    IF index = 0 THEN
        RETURN;
    END_IF
END_IF
IF NOT _M_CaptureConfig(SetName := '_validation', Kind := Info.Kind, ModelIndex := index) THEN
    RETURN;
END_IF
IF NOT _M_ValidateSetShape(Store := _loadSnapshot, Info := Info, AnyRevision := TRUE) THEN
    RETURN;
END_IF
IF NOT _M_OpenModelView(Index := index) THEN
    RETURN;
END_IF
_M_LiveApply := _M_ApplySet(SetName := Info.SetName, RecordCount := Info.RecordCount,
    Kind := Info.Kind, Restoring := TRUE);
IF _M_LiveApply AND (Info.Kind = E_ConfigKind.PAR_CFG) THEN
    _M_LiveApply := _M_SaveModelData();
END_IF
_pModelView := 0;
END_METHOD

// AvailableModels index of a model code, 0 when the catalog does not offer it.
METHOD PRIVATE _M_ModelIndexOf : UDINT
VAR_INPUT
    ModelCode : STRING(64);
END_VAR
VAR
    i : INT;
END_VAR
_M_ModelIndexOf := 0;
IF ModelCode = '' THEN
    RETURN;
END_IF
FOR i := 1 TO AvailableModelCount DO
    IF AvailableModels[i].ModelCode = ModelCode THEN
        _M_ModelIndexOf := INT_TO_UDINT(i);
        RETURN;
    END_IF
END_FOR
END_METHOD

// §3.8b — "restore is fail-closed and never silent". Every module that ran
// M_RestoreStationCfg and found an unrecognized image is holding one report;
// this takes them and annunciates each with the OWNING module's canonical path,
// which is what makes the message actionable instead of "something was lost".
//
// The event is AUTO_RESET and therefore never blocking: the consequence belongs
// to E_ConfigRestorePolicy, evaluated in ReleaseReportStart, so a station that
// declared DEFAULTS_AND_ANNUNCIATE really does run while the annunciation
// stands. It stays open until an ENGINEER acknowledges it, because nothing
// makes a lost image come back and an event that closed itself would be a lie.
METHOD PRIVATE _M_DrainRestoreLoss
VAR
    guard    : INT;
    path     : STRING(80);
    expected : UINT;
    found    : UINT;
END_VAR
// §7.7(c) - the local user table is retained outside the module walk; its loss
// is announced and acknowledged exactly like a module's.
IF Access.M_TakeRestoreLoss() THEN
    path := CONCAT(_name, '.Access');
    _M_AnnounceRestoreLoss(Path := path, Text := 'std.error.accessRestoreLost');
END_IF
// Bounded per scan (§5.6): losses are one-shot, so a large subtree simply
// finishes draining over the next few scans instead of stretching one.
FOR guard := 1 TO PL_Fraktal.MAX_EM_CHILDREN DO
    IF NOT M_TakeRestoreLoss(Path => path, Expected => expected, Found => found) THEN
        RETURN;
    END_IF
    _M_AnnounceRestoreLoss(Path := path, Text := 'std.error.configRestoreLost');
END_FOR
END_METHOD

// §3.8b - publish one lost image and open (or extend) its annunciation.
METHOD PRIVATE _M_AnnounceRestoreLoss
VAR_INPUT
    Path : STRING(80);
    Text : STRING(80);
END_VAR
ConfigPersist.RestoreLost := TRUE;
ConfigPersist.RestoreAcknowledged := FALSE;
ConfigPersist.LostPath := Path;
IF _restoreEvt = 0 THEN
    _restoreEvt := AlarmLog.Raise(Reason := E_Reason.CONFIG_RESTORE_LOST,
        Text := Text, Source := Path,
        Severity := E_Severity.MED, Category := E_Category.SYSTEM,
        ResetClass := E_ResetClass.AUTO_RESET);
ELSE
    // A second losing owner gets its own ring entry: a summary that named only
    // the first would hide the rest of the damage.
    _M_RaiseMaintenance(Reason := E_Reason.CONFIG_RESTORE_LOST, Text := Text);
END_IF
END_METHOD

// §3.8b — an operator of at least ENGINEER level accepts that a configuration
// image was lost. Under BLOCK_UNTIL_ACKNOWLEDGED this is what releases
// START_STOP again; under DEFAULTS_AND_ANNUNCIATE it is what clears the
// standing annunciation.
//
// The level is checked directly rather than through a gated action, because
// §3.8b names ENGINEER specifically and a station may legitimately have left
// DATA_WRITE or CONFIG_SET open to a lower level. Acknowledging a lost
// commissioning is a different decision from editing a value.
METHOD AcknowledgeConfigRestore : BOOL
AcknowledgeConfigRestore := FALSE;
IF Access.CurrentLevel < E_AccessLevel.ENGINEER THEN
    RETURN;
END_IF
IF NOT ConfigPersist.RestoreLost THEN
    RETURN;                                // nothing to acknowledge
END_IF
ConfigPersist.RestoreAcknowledged := TRUE;
IF _restoreEvt > 0 THEN
    AlarmLog.Gone(Slot := _restoreEvt);
    _restoreEvt := 0;
END_IF
Access.RecordActivity();
AcknowledgeConfigRestore := TRUE;
END_METHOD

// §3.8b — refuse a set operation, naming the offending record. "One rejection
// aborts the whole load naming the offending (Scope, WriteKey)": a refusal that
// says only "rejected" leaves an engineer diffing two machines by hand.
METHOD PRIVATE _M_RejectConfigSet
VAR_INPUT
    Scope : STRING(80);
    Key   : STRING(160);
END_VAR
ConfigPersist.LastRejectScope := Scope;
ConfigPersist.LastRejectKey := Key;
_M_RaiseMaintenance(Reason := E_Reason.CONFIG_SET_REJECTED,
    Text := 'std.error.configSetRejected');
END_METHOD

// §3.8b — the gate every set operation shares: CONFIG_SET (never DATA_WRITE —
// replacing a machine's entire parametrization is not the same decision as
// changing one number), a wired store, and the owning root READY.
METHOD PRIVATE _M_SetOpAllowed : BOOL
_M_SetOpAllowed := FALSE;
IF NOT _M_ConfigRestored() THEN
    RETURN;
END_IF
IF NOT Access.PermitsLogged(Gate := E_GatedAction.CONFIG_SET) THEN
    RETURN;
END_IF
IF _configStore = 0 THEN
    RETURN;
END_IF
IF _exec <> E_ExecState.READY THEN
    RETURN;
END_IF
_M_SetOpAllowed := TRUE;
END_METHOD

// §3.8b - remove a named set. Gated exactly like save and load (CONFIG_SET, a
// wired store, the root READY) because removing somebody's commissioned set is
// the same order of decision as replacing it, and audited with the set name.
// A store that has held MAX_CONFIG_SETS names needs this to hold a new one.
METHOD DeleteConfigSet : BOOL
VAR_INPUT
    SetName : STRING(80);
END_VAR
DeleteConfigSet := FALSE;
ConfigPersist.LastSetName := SetName;
ConfigPersist.LastSetRecords := 0;
IF NOT _M_SetOpAllowed() THEN
    RETURN;
END_IF
IF NOT _configStore.M_Delete(SetName := SetName) THEN
    RETURN;
END_IF
DeleteConfigSet := TRUE;
// The store's retained memory changed; not durable until written out.
_M_MarkPersistPending();
ListConfigSets();                          // the published listing follows
END_METHOD

// §3.8d - the effective level to read or write one registered value, from
// what its owning module declared and this root's policy. The root's own
// framework keys (unit.modePolicy.*) are in the built-in class. An unknown key
// resolves to ADMIN: the write path refuses it anyway, and a level check must
// never be the thing that lets an unknown key through.
METHOD PRIVATE _M_DataLevelOf : E_AccessLevel
VAR_INPUT
    TargetPath : STRING(255);
    WriteKey   : STRING(160);
    ForWrite   : BOOL;
END_VAR
VAR
    grant    : ST_ConfigAccess;
    minLevel : E_AccessLevel;
END_VAR
_M_DataLevelOf := E_AccessLevel.ADMIN;
IF (TargetPath = Status.Name) AND (LEFT(WriteKey, 16) = 'unit.modePolicy.') THEN
    _M_DataLevelOf := Access.M_DataLevel(ClassId := '', MinLevel := E_AccessLevel.NONE,
        ForWrite := ForWrite);
    RETURN;
END_IF
IF NOT M_ConfigAccessOf(Scope := TargetPath, WriteKey := WriteKey, Grant := grant) THEN
    RETURN;
END_IF
IF ForWrite THEN
    minLevel := grant.MinWriteLevel;
ELSE
    minLevel := grant.MinReadLevel;
END_IF
_M_DataLevelOf := Access.M_DataLevel(ClassId := grant.ClassId, MinLevel := minLevel,
    ForWrite := ForWrite);
END_METHOD

// §3.8d - declare a project data class on this root, at Setup. The levels are
// defaults: a class the deployment already edited keeps its persisted levels.
METHOD M_DeclareDataClass : BOOL
VAR_INPUT
    ClassId    : STRING(80);
    LabelKey   : STRING(160);
    ReadLevel  : E_AccessLevel;
    WriteLevel : E_AccessLevel;
END_VAR
M_DeclareDataClass := Access.M_DeclareClass(ClassId := ClassId,
    LabelKey := LabelKey, ReadLevel := ReadLevel, WriteLevel := WriteLevel);
END_METHOD

// §3.8d/§7.7(b) - edit a class's read or write level. The same gate as
// every other policy edit (ACCESS_POLICY), audited through the mailbox.
METHOD SetDataClassLevel : BOOL
VAR_INPUT
    ClassId  : STRING(160);
    Level    : DINT;
    ForWrite : BOOL;
END_VAR
VAR
    levelReq : E_AccessLevel;
END_VAR
SetDataClassLevel := FALSE;
IF NOT Access.PermitsLogged(Gate := E_GatedAction.ACCESS_POLICY) THEN
    RETURN;
END_IF
IF (Level < TO_DINT(E_AccessLevel.NONE)) OR (Level > TO_DINT(E_AccessLevel.ADMIN))
OR (LEN(ClassId) > 40) THEN
    RETURN;
END_IF
levelReq := Level;                          // range-checked above
SetDataClassLevel := Access.M_SetClassLevel(ClassId := ClassId,
    Level := levelReq, ForWrite := ForWrite);
IF SetDataClassLevel THEN
    ConfigRev := ConfigRev + 1;             // every manifest level may have moved
END_IF
END_METHOD

// §3.8e - TRUE when a (Scope, WriteKey) the subtree did not own names a value of
// the line this Unit references: the line is published under this Unit's own
// scope, and its keys alone begin 'line.'.
METHOD PRIVATE _M_IsLineKey : BOOL
VAR_INPUT
    Scope    : STRING(255);
    WriteKey : STRING(160);
END_VAR
_M_IsLineKey := (_pLine <> 0) AND (Scope = Status.Name)
    AND (LEFT(WriteKey, 5) = 'line.');
END_METHOD

// §3.8e - the subtree first; a line key it does not own goes to the line.
METHOD M_ApplyConfigWrite : BOOL
VAR_INPUT
    Scope     : STRING(255);
    WriteKey  : STRING(160);
    Revision  : UDINT;
    TextValue : STRING(255);
    RootReady : BOOL;
END_VAR
M_ApplyConfigWrite := SUPER^.M_ApplyConfigWrite(Scope := Scope,
    WriteKey := WriteKey, Revision := Revision, TextValue := TextValue,
    RootReady := RootReady);
IF (NOT M_ApplyConfigWrite) AND _M_IsLineKey(Scope := Scope, WriteKey := WriteKey) THEN
    M_ApplyConfigWrite := _pLine^.M_ApplyConfigWrite(Scope := _pLine^.Status.Name,
        WriteKey := WriteKey, Revision := Revision, TextValue := TextValue,
        RootReady := RootReady);
END_IF
END_METHOD

// §3.8e - the staging walk is the write walk, line leg included.
METHOD M_StageConfigWrite : BOOL
VAR_INPUT
    Scope     : STRING(255);
    WriteKey  : STRING(160);
    Revision  : UDINT;
    TextValue : STRING(255);
    RootReady : BOOL;
END_VAR
M_StageConfigWrite := SUPER^.M_StageConfigWrite(Scope := Scope,
    WriteKey := WriteKey, Revision := Revision, TextValue := TextValue,
    RootReady := RootReady);
IF (NOT M_StageConfigWrite) AND _M_IsLineKey(Scope := Scope, WriteKey := WriteKey) THEN
    M_StageConfigWrite := _pLine^.M_StageConfigWrite(Scope := _pLine^.Status.Name,
        WriteKey := WriteKey, Revision := Revision, TextValue := TextValue,
        RootReady := RootReady);
END_IF
END_METHOD

// §3.8e - the capture walk is the write walk, line leg included.
METHOD M_ApplyCapture : BOOL
VAR_INPUT
    Scope     : STRING(255);
    WriteKey  : STRING(160);
    Revision  : UDINT;
    RootReady : BOOL;
END_VAR
M_ApplyCapture := SUPER^.M_ApplyCapture(Scope := Scope, WriteKey := WriteKey,
    Revision := Revision, RootReady := RootReady);
IF (NOT M_ApplyCapture) AND _M_IsLineKey(Scope := Scope, WriteKey := WriteKey) THEN
    M_ApplyCapture := _pLine^.M_ApplyCapture(Scope := _pLine^.Status.Name,
        WriteKey := WriteKey, Revision := Revision, RootReady := RootReady);
END_IF
END_METHOD

// §3.8e/§3.8d - the access walk is the write walk, line leg included, so a line
// value is checked against the level the line declared for it.
METHOD M_ConfigAccessOf : BOOL
VAR_INPUT
    Scope    : STRING(255);
    WriteKey : STRING(160);
END_VAR
VAR_IN_OUT
    Grant : ST_ConfigAccess;
END_VAR
M_ConfigAccessOf := SUPER^.M_ConfigAccessOf(Scope := Scope, WriteKey := WriteKey,
    Grant := Grant);
IF (NOT M_ConfigAccessOf) AND _M_IsLineKey(Scope := Scope, WriteKey := WriteKey) THEN
    M_ConfigAccessOf := _pLine^.M_ConfigAccessOf(Scope := _pLine^.Status.Name,
        WriteKey := WriteKey, Grant := Grant);
END_IF
END_METHOD

// Core §3.8a - declare this root's own recipe record (its ParCfg) and the
// provider it is loaded from. The PAR_CFG values registered inside it become
// editable for EVERY model the root offers (AvailableModels), not only the
// active one, and an edit is written back to the provider's record so a
// changeover keeps it - when the provider is also an I_RecipeStore.
METHOD M_RegisterModelData : BOOL
VAR_INPUT
    pData     : PVOID;
    Size      : UDINT;
    RecipeKey : STRING(80);
    Provider  : I_RecipeProvider;
END_VAR
M_RegisterModelData := FALSE;
IF (pData = 0) OR (Size = 0) OR (Size > PL_Fraktal.MAX_MODEL_DATA_BYTES)
OR (RecipeKey = '') OR (Provider = 0) THEN
    RETURN;
END_IF
_modelProvider := Provider;
__QUERYINTERFACE(Provider, _modelCatalog);
_modelKey := RecipeKey;
M_RegisterModelData := _M_SetModelRegion(pRegion := pData, Size := Size);
END_METHOD

// Serve model-scoped values of AvailableModels[Index] for this one request. 0,
// or the active model's index, is the live record and opens nothing. The record
// is loaded over a copy of the live one, so the provider's SchemaVersion check
// compares like with like. FALSE = no such model, or its record did not load.
METHOD PRIVATE _M_OpenModelView : BOOL
VAR_INPUT
    Index : UDINT;
END_VAR
_M_OpenModelView := FALSE;
_pModelView := 0;
_viewModelCode := '';
IF Index = 0 THEN
    _M_OpenModelView := TRUE;
    RETURN;
END_IF
IF (_modelProvider = 0) OR (_pModelRegion = 0)
OR (Index > TO_UDINT(AvailableModelCount)) THEN
    RETURN;
END_IF
IF AvailableModels[Index].ModelCode = Model.ModelCode THEN
    _M_OpenModelView := TRUE;              // the active model: its record is live
    RETURN;
END_IF
MEMCPY(destAddr := ADR(_modelBuf), srcAddr := _pModelRegion, n := _modelRegionSize);
IF NOT _modelProvider.Load(ModelCode := AvailableModels[Index].ModelCode,
        RecipeKey := _modelKey, pParCfg := ADR(_modelBuf), Size := _modelRegionSize) THEN
    RETURN;
END_IF
_viewModelCode := AvailableModels[Index].ModelCode;
_pModelView := ADR(_modelBuf);
_M_OpenModelView := TRUE;
END_METHOD

// §3.8a - WriteConfig for the model AvailableModels[ModelIndex] (0 = the active
// model). A model-data value is stored in that model's record and saved back to
// the provider; any other value is written as WriteConfig writes it.
METHOD WriteModelConfig : BOOL
VAR_INPUT
    ModelIndex : UDINT;
    TargetPath : STRING(255);
    WriteKey   : STRING(160);
    Revision   : DINT;
    TextValue  : STRING(255);
END_VAR
WriteModelConfig := FALSE;
IF NOT _M_OpenModelView(Index := ModelIndex) THEN
    RETURN;
END_IF
WriteModelConfig := WriteConfig(TargetPath := TargetPath, WriteKey := WriteKey,
    Revision := Revision, TextValue := TextValue);
_pModelView := 0;
END_METHOD

// §3.8a - the manifest walk (M_AppendConfig) with the model-data values of
// AvailableModels[ModelIndex] (0 = the active model). FALSE = no such model.
// For another model the walk yields that model's data only: the rest of the
// manifest is the running station's and is served by index 0.
METHOD M_AppendModelConfig : BOOL
VAR_INPUT
    Pager      : REFERENCE TO FB_ConfigPager;
    ModelIndex : UDINT;
END_VAR
M_AppendModelConfig := FALSE;
IF NOT _M_OpenModelView(Index := ModelIndex) THEN
    RETURN;
END_IF
Pager.M_SetModelOnly(Enabled := ModelIndex > 0);
M_AppendConfig(Pager := Pager);
Pager.M_SetModelOnly(Enabled := FALSE);
_pModelView := 0;
M_AppendModelConfig := TRUE;
END_METHOD

// Write the record a model-scoped value was just stored into back to the
// provider: the viewed model's buffer, or the live record for the active model.
METHOD PRIVATE _M_SaveModelData : BOOL
VAR
    store : I_RecipeStore;
END_VAR
_M_SaveModelData := FALSE;
IF _modelProvider = 0 THEN
    RETURN;
END_IF
IF NOT __QUERYINTERFACE(_modelProvider, store) THEN
    RETURN;
END_IF
IF _pModelView <> 0 THEN
    _M_SaveModelData := store.Save(ModelCode := _viewModelCode, RecipeKey := _modelKey,
        pData := _pModelView, Size := _modelRegionSize);
ELSE
    _M_SaveModelData := store.Save(ModelCode := Model.ModelCode, RecipeKey := _modelKey,
        pData := _pModelRegion, Size := _modelRegionSize);
END_IF
END_METHOD

// §3.8e/§8.5.2 - reference the line this root belongs to (owner or mirror, on
// this controller). A Unit references at most one line; 0 detaches it.
METHOD SetLine : BOOL
VAR_INPUT
    pLine : POINTER TO FB_LineData;
END_VAR
_pLine := pLine;
_lineHost := FALSE;
IF pLine <> 0 THEN
    // The first root to reference a line hosts it (ticks it, lends its log); a
    // line is never a child, so nothing else would run it (§3.8e(a)).
    _lineHost := pLine^.M_BindHost(pHost := THIS, pAlarmLog := ADR(AlarmLog));
END_IF
_shiftInit := FALSE;
CurrentShift := 0;
SetLine := (pLine <> 0);
END_METHOD

// Evaluate only at a finite boundary, or after an empty-calendar edit.
METHOD M_ShiftTick : BOOL
VAR_INPUT
    Now : DT;
    Synchronized : BOOL;
END_VAR
VAR
    idx : INT;
    started : DT;
    ending : DT;
    target : UDINT;
    crossed : BOOL;
    quality : BOOL;
END_VAR
M_ShiftTick := FALSE;
IF _pLine = 0 THEN CurrentShift := 0; ShiftProductionTarget := 0; RETURN; END_IF
IF _shiftInit THEN
    IF Now < _shiftLastNow THEN _shiftSync := FALSE; END_IF
    _shiftLastNow := Now;
    IF (_shiftEnd <> DT#1970-01-01-00:00:00) AND (Now < _shiftEnd) THEN RETURN; END_IF
    IF Now < ShiftStartedAt THEN RETURN; END_IF // no negative history after a backward jump
    IF (_shiftEnd = DT#1970-01-01-00:00:00)
    AND (_shiftCalendarRev = _pLine^.OutImm.Revision) THEN RETURN; END_IF
END_IF
IF NOT _pLine^.M_ShiftInterval(Now := Now, ShiftIndex => idx,
        StartAt => started, EndAt => ending, Target => target) THEN
    _shiftSync := FALSE; RETURN;
END_IF
crossed := _shiftInit AND (_shiftEnd <> DT#1970-01-01-00:00:00);
IF _shiftInit AND NOT crossed AND (idx = 0) THEN
    // Empty/off interval continues; an edit must not erase accrued production.
    _shiftEnd := ending;
    _shiftCalendarRev := _pLine^.OutImm.Revision;
    RETURN;
END_IF
IF _shiftInit THEN
    quality := Synchronized;
    IF crossed AND (DT_TO_UDINT(Now) > DT_TO_UDINT(_shiftEnd) + 1) THEN quality := FALSE; END_IF
    _M_CloseShift(Now := Now, Synchronized := quality);
    M_ShiftTick := TRUE;
END_IF
_shiftInit := TRUE;
CurrentShift := idx;
ShiftStartedAt := Now; // observed start, never invent production before attachment/jump
ShiftProductionTarget := target;
_shiftEnd := ending;
_shiftLastNow := Now;
_shiftCalendarRev := _pLine^.OutImm.Revision;
_shiftSync := Synchronized;
_shiftManualReset := FALSE;
END_METHOD

// §8.5.2(b) - one operation in one scan: record the ending shift as its figures stood,
// then reset the per-shift counts and OEE accumulators (the trend ring is kept). A
// boundary on an unsynchronized clock still closes - stopping the accounting would
// lose more than a late boundary does - and the record says so.
METHOD PRIVATE _M_CloseShift
VAR_INPUT
    Now          : DT;
    Synchronized : BOOL;
END_VAR
VAR
    i         : INT;
    auditSlot : INT;
END_VAR
_M_OeeCompute(); // capture current factors before counters are cleared
FOR i := PL_Fraktal.MAX_SHIFT_HISTORY TO 2 BY -1 DO
    ShiftHistory[i] := ShiftHistory[i - 1];
END_FOR
IF ShiftHistoryCount >= PL_Fraktal.MAX_SHIFT_HISTORY THEN
    ShiftHistoryTruncated := TRUE;
ELSE
    ShiftHistoryCount := ShiftHistoryCount + 1;
END_IF
ShiftHistory[1].SchemaVersion := 3;
ShiftHistory[1].ProductionTarget := ShiftProductionTarget;
ShiftHistory[1].ShiftIndex := CurrentShift;
ShiftHistory[1].StartAt := ShiftStartedAt;
ShiftHistory[1].EndAt := Now;
ShiftHistory[1].TimeSynchronized := _shiftSync AND Synchronized;
ShiftHistory[1].ManualReset := _shiftManualReset;
ShiftHistory[1].GoodCount := GoodCount;
ShiftHistory[1].NokCount := NokCount;
ShiftHistory[1].ReworkCount := ReworkCount;
ShiftHistory[1].RunMs := Oee.RunMs;
ShiftHistory[1].DownMs := Oee.DownMs;
ShiftHistory[1].IdleMs := Oee.IdleMs;
ShiftHistory[1].Availability := Oee.Availability;
ShiftHistory[1].AvailValid := Oee.AvailValid;
ShiftHistory[1].Performance := Oee.Performance;
ShiftHistory[1].PerfValid := Oee.PerfValid;
ShiftHistory[1].Quality := Oee.Quality;
ShiftHistory[1].QualValid := Oee.QualValid;
ShiftHistory[1].Oee := Oee.Oee;
ShiftHistory[1].OeeValid := Oee.OeeValid;
_oeeGoodBase := 0;
_oeeNokBase := 0;
GoodCount := 0;
NokCount := 0;
ReworkCount := 0;
Oee.RunMs := 0;
Oee.DownMs := 0;
Oee.IdleMs := 0;
_M_OeeCompute();
auditSlot := AlarmLog.Raise(Reason := E_Reason.NONE, Text := 'std.audit.shiftClosed',
    Source := _name, Severity := E_Severity.LOW, Category := E_Category.SYSTEM,
    ResetClass := E_ResetClass.AUTO_RESET);
IF auditSlot > 0 THEN
    AlarmLog.Gone(Slot := auditSlot);    // come+gone: into the ring and the event sink
END_IF
END_METHOD

// §3.8b — save the current parametrization as a named set.
//
// The set is a PROJECTION of the same deterministic walk that builds the
// §3.10.2 manifest: M_AppendConfig runs exactly as a QUERY_CONFIG would run it,
// and the pager files every capability of the requested ConfigKind as a
// (Scope, WriteKey) record. There is no second enumeration of "what this
// station's configuration consists of" to drift from the first (§1.1 O9).
//
// Kind selects which of the two kinds of set this is: STATION_CFG for a station
// set (deployment data), PAR_CFG for a model set (one model's recipe data).
METHOD SaveConfigSet : BOOL
VAR_INPUT
    SetName : STRING(80);
    Kind    : E_ConfigKind;
END_VAR
VAR
    info    : ST_ConfigSetInfo;
    records : INT;
END_VAR
SaveConfigSet := FALSE;
ConfigPersist.LastSetName := SetName;
ConfigPersist.LastSetRecords := 0;
IF NOT _M_SetOpAllowed() THEN
    RETURN;
END_IF
IF SetName = '' THEN
    RETURN;
END_IF
info.Used := TRUE;
info.SetName := SetName;
info.RootIdentity := Status.Name;
info.SetSchema := CONFIG_SET_SCHEMA;
info.ConfigRev := ConfigRev;
info.Kind := Kind;
IF Kind = E_ConfigKind.PAR_CFG THEN
    info.ModelCode := Model.ModelCode;     // a model set belongs to ONE model
ELSE
    info.ModelCode := '';
END_IF
info.RecordCount := 0;
info.CreatedAt := F_Now();
info.TimeSynchronized := F_TimeSynchronized();
IF NOT _configPager.M_SetupSetSave(Store := _configStore, Info := info) THEN
    RETURN;
END_IF
M_AppendConfig(Pager := _configPager);     // the SAME walk as the manifest
SaveConfigSet := _configPager.M_FinishSetSave(Records => records);
ConfigPersist.LastSetRecords := records;
IF SaveConfigSet THEN
    // The set now lives in the store's retained memory, which is not durable
    // until it is written out - the same promise as any other accepted write.
    _M_MarkPersistPending();
END_IF
END_METHOD

// §3.8b — apply a named set. STAGED and ALL-OR-NOTHING.
//
// Pass 1 validates every record through its owning module's typed handler and
// changes nothing. Only if all of them pass does pass 2 apply them. A
// half-applied machine parametrization is never a valid outcome, and the only
// way to guarantee that is to know the answer for every record before touching
// the first one.
//
// A record whose capability no longer exists fails pass 1 like any other and is
// REPORTED by name - never silently dropped, because a set that quietly skipped
// the one value that mattered restores a machine to almost its commissioned
// state, which is the failure that is hardest to notice.
METHOD LoadConfigSet : BOOL
VAR_INPUT
    SetName : STRING(80);
END_VAR
VAR
    info    : ST_ConfigSetInfo;
END_VAR
LoadConfigSet := FALSE;
ConfigPersist.LastSetName := SetName;
ConfigPersist.LastSetRecords := 0;
ConfigPersist.LastRejectScope := '';
ConfigPersist.LastRejectKey := '';
IF NOT _M_SetOpAllowed() THEN
    RETURN;
END_IF
IF NOT _M_CopySet(SetName := SetName) THEN
    RETURN;
END_IF
IF NOT _loadSnapshot.M_ReadInfo(SetName := SetName, Info := info) THEN
    _M_RejectConfigSet(Scope := '', Key := SetName);
    RETURN;
END_IF
IF info.RootIdentity <> Status.Name THEN
    // The set carries the identity of the root that produced it precisely so
    // this can be asked. Every record's Scope is prefixed by that identity, so
    // a mismatch would fail record by record anyway - naming the root instead
    // tells the operator WHY in one line.
    _M_RejectConfigSet(Scope := info.RootIdentity, Key := '');
    RETURN;
END_IF
IF info.Kind = E_ConfigKind.PAR_CFG THEN
    // §3.8b: a MODEL set "shall be applied through the §3.8 changeover
    // transaction (PrepareRecipe -> recursive readiness -> infallible
    // CommitRecipe), never as a sequence of per-field writes". Applying it here
    // would be exactly that forbidden sequence, so it is refused. Saving a
    // model set is supported; loading one is a changeover this build does not
    // implement, and refusing is the honest half of that.
    _M_RejectConfigSet(Scope := info.ModelCode, Key := '');
    RETURN;
END_IF
IF NOT _M_CaptureConfig(SetName := '_validation', Kind := info.Kind, ModelIndex := 0) THEN RETURN; END_IF
IF NOT _M_ValidateSetShape(Store := _loadSnapshot, Info := info, AnyRevision := FALSE) THEN
    RETURN;
END_IF
IF NOT _M_ApplySet(SetName := SetName, RecordCount := info.RecordCount, Kind := info.Kind,
        Restoring := FALSE) THEN
    RETURN;
END_IF
ConfigRev := ConfigRev + 1;
ConfigPersist.LastSetRecords := info.RecordCount;
_M_MarkPersistPending();
_M_RaiseMaintenance(Reason := E_Reason.EVENT_CONFIG_SET_APPLIED,
    Text := 'std.audit.configSetApplied');
LoadConfigSet := TRUE;
END_METHOD

// §3.8b - replay the set frozen in _loadSnapshot. STAGED and ALL-OR-NOTHING:
// pass 1 validates every record through its owning module's typed handler and
// changes nothing; only if all of them pass does pass 2 apply them. A record
// whose capability no longer exists fails pass 1 like any other and is named.
//
// Shared by an operator's LoadConfigSet and the start-up restore of the live
// documents. Restoring skips the session's per-value level (§3.8d(e)): those
// values were accepted once already, and replaying them is the machine's act,
// not an operator's. With a model view open the values go to that record.
METHOD PRIVATE _M_ApplySet : BOOL
VAR_INPUT
    SetName     : STRING(80);
    RecordCount : INT;
    Kind        : E_ConfigKind;
    Restoring   : BOOL;
END_VAR
VAR
    record    : ST_ConfigRecord;
    i         : INT;
    applied   : BOOL;
    lineBatch : BOOL;
END_VAR
_M_ApplySet := FALSE;
lineBatch := (Kind = E_ConfigKind.LINE_CFG) AND (_pLine <> 0);
IF lineBatch THEN
    IF NOT _pLine^.M_BeginConfigBatch() THEN RETURN; END_IF
END_IF
// ---- pass 1: stage. Nothing in the machine changes in this loop. ----
FOR i := 1 TO RecordCount DO
    IF NOT _loadSnapshot.M_ReadRecord(SetName := SetName, Index := i,
            Record := record) THEN
        _M_RejectConfigSet(Scope := '', Key := SetName);
        IF lineBatch THEN _pLine^.M_EndConfigBatch(); END_IF
        RETURN;
    END_IF
    // §3.8d(e) - CONFIG_SET alone cannot replace a value this session could
    // not edit one at a time. Checked in the staging pass, so nothing moved.
    IF NOT Restoring THEN
        IF NOT Access.M_PermitsLevelLogged(Required := _M_DataLevelOf(TargetPath := record.Scope,
                WriteKey := record.WriteKey, ForWrite := TRUE)) THEN
            _M_RejectConfigSet(Scope := record.Scope, Key := record.WriteKey);
            IF lineBatch THEN _pLine^.M_EndConfigBatch(); END_IF
            RETURN;
        END_IF
    END_IF
    IF NOT _M_StageOneRecord(Record := record) THEN
        _M_RejectConfigSet(Scope := record.Scope, Key := record.WriteKey);
        IF lineBatch THEN _pLine^.M_EndConfigBatch(); END_IF
        RETURN;
    END_IF
END_FOR
IF lineBatch THEN
    IF NOT _pLine^.M_ValidateConfigBatch() THEN
        _pLine^.M_EndConfigBatch(); _M_RejectConfigSet(Scope := Status.Name, Key := SetName); RETURN;
    END_IF
END_IF
// ---- pass 2: apply. Every record already proved acceptable on the SAME
// validator, so a refusal here cannot be a data problem. ----
FOR i := 1 TO RecordCount DO
    IF NOT _loadSnapshot.M_ReadRecord(SetName := SetName, Index := i,
            Record := record) THEN
        IF lineBatch THEN _pLine^.M_EndConfigBatch(); END_IF
        _M_ConfigSetHalfApplied(Scope := record.Scope, Key := record.WriteKey);
        RETURN;
    END_IF
    applied := _M_WriteBaseConfig(TargetPath := record.Scope,
        WriteKey := record.WriteKey, Revision := record.Revision,
        TextValue := record.ValueText, Commit := TRUE);
    IF NOT applied THEN
        applied := M_ApplyConfigWrite(Scope := record.Scope,
            WriteKey := record.WriteKey, Revision := record.Revision,
            TextValue := record.ValueText,
            RootReady := (_exec = E_ExecState.READY) OR (_pModelView <> 0));
    END_IF
    IF NOT applied THEN
        IF lineBatch THEN _pLine^.M_EndConfigBatch(); END_IF
        _M_ConfigSetHalfApplied(Scope := record.Scope, Key := record.WriteKey);
        RETURN;
    END_IF
END_FOR
IF lineBatch THEN
    _pLine^.M_CommitConfigBatch();
END_IF
_M_ApplySet := TRUE;
END_METHOD

// §3.8b — would this record be accepted? The same two-step the write path
// takes: framework-owned keys first, then the recursive walk to the owning
// module. Sharing the writers' own code with Commit := FALSE is what makes
// "staged" mean something: a separate validator could pass a record the write
// path would then refuse, and the load would be half-applied after all.
METHOD PRIVATE _M_StageOneRecord : BOOL
VAR_INPUT
    Record : ST_ConfigRecord;
END_VAR
_M_StageOneRecord := _M_WriteBaseConfig(TargetPath := Record.Scope,
    WriteKey := Record.WriteKey, Revision := Record.Revision,
    TextValue := Record.ValueText, Commit := FALSE);
IF _M_StageOneRecord THEN
    RETURN;
END_IF
_M_StageOneRecord := M_StageConfigWrite(Scope := Record.Scope,
    WriteKey := Record.WriteKey, Revision := Record.Revision,
    TextValue := Record.ValueText,
    // Another model's record is not what the machine is running on.
    RootReady := (_exec = E_ExecState.READY) OR (_pModelView <> 0));
END_METHOD

// §3.8b — a record passed staging and then failed to apply. This cannot
// happen: both run the same validator on the same data in the same scan. If it
// ever does, the machine is half-parametrized and that is a state the standard
// says is never valid - so it is escalated as a BLOCKING alarm rather than
// returned as a FALSE somebody might retry. A framework defect that leaves a
// machine half-configured has to stop it, not inconvenience it.
METHOD PRIVATE _M_ConfigSetHalfApplied
VAR_INPUT
    Scope : STRING(80);
    Key   : STRING(160);
END_VAR
ConfigPersist.LastRejectScope := Scope;
ConfigPersist.LastRejectKey := Key;
AlarmLog.Raise(Reason := E_Reason.CONFIG_SET_REJECTED,
    Text := 'std.error.configSetHalfApplied', Source := Scope,
    Severity := E_Severity.HIGH, Category := E_Category.SYSTEM,
    ResetClass := E_ResetClass.MANUAL_RESET);
END_METHOD

// §3.8b — refresh the published listing of stored sets. Read-only, so it is
// gated on CONFIG_SET without the audited write path: seeing which sets exist
// is not replacing a machine's parametrization.
METHOD ListConfigSets : BOOL
VAR
    i     : INT;
    total : INT;
END_VAR
ListConfigSets := FALSE;
FOR i := 1 TO PL_Fraktal.MAX_CONFIG_SETS DO
    ConfigSets[i].Used := FALSE;
    ConfigSets[i].SetName := '';
    ConfigSets[i].RecordCount := 0;
END_FOR
ConfigSetCount := 0;
IF NOT Access.Permits(Gate := E_GatedAction.CONFIG_SET) THEN
    RETURN;
END_IF
IF _configStore = 0 THEN
    RETURN;
END_IF
total := _configStore.M_Count();
FOR i := 1 TO PL_Fraktal.MAX_CONFIG_SETS DO
    IF i > total THEN
        EXIT;
    END_IF
    IF _configStore.M_InfoAt(Index := i, Info := ConfigSets[i]) THEN
        ConfigSetCount := i;
    END_IF
END_FOR
ListConfigSets := TRUE;
END_METHOD

// §3.8b — serve one line of a set's JSON document. Line 0 is the header and
// 1..RecordCount are the records, so a client pulls a movable document a line
// at a time and no full document buffer ever exists in the PLC - the same
// paging discipline QUERY_CONFIG already uses for the manifest.
//
// This is what makes a set MOVABLE, which is the point of naming sets at all: a
// station's commissioning can leave the controller as text, be reviewed,
// diffed, version-controlled and put on the next machine.
METHOD ExportConfigSetLine : BOOL
VAR_INPUT
    SetName : STRING(80);
    Line    : INT;
END_VAR
VAR
    info   : ST_ConfigSetInfo;
    record : ST_ConfigRecord;
END_VAR
ExportConfigSetLine := FALSE;
ConfigSetDocument := '';
ConfigSetDocumentLine := Line;
ConfigSetDocumentLines := 0;
IF NOT Access.Permits(Gate := E_GatedAction.CONFIG_SET) THEN
    RETURN;
END_IF
IF _configStore = 0 THEN
    RETURN;
END_IF
IF NOT _configStore.M_ReadInfo(SetName := SetName, Info := info) THEN
    RETURN;
END_IF
ConfigSetDocumentLines := info.RecordCount;
IF Line <= 0 THEN
    ConfigSetDocument := _setJson.M_Header(Info := info);
ELSE
    IF NOT _configStore.M_ReadRecord(SetName := SetName, Index := Line,
            Record := record) THEN
        RETURN;
    END_IF
    IF NOT Access.M_PermitsLevel(Required := _M_DataLevelOf(TargetPath := record.Scope,
            WriteKey := record.WriteKey, ForWrite := FALSE)) THEN
        RETURN;                           // §3.8d(e): the export fails, it is not thinned
    END_IF
    ConfigSetDocument := _setJson.M_Record(Record := record);
END_IF
// An empty line means the projection REFUSED to render it rather than shorten
// it, so the export fails here instead of shipping a document with a hole.
ExportConfigSetLine := (ConfigSetDocument <> '');
END_METHOD

// §3.8b — take one line of a set's JSON document back in. A header line opens
// a store save, record lines append to it, and Commit closes it.
//
// Import writes into the STORE, never into the machine. Bringing a document in
// and applying it to the equipment are two decisions, and keeping them apart is
// what lets LoadConfigSet stay staged and all-or-nothing: an imported set is
// validated against THIS machine's capabilities when somebody chooses to load
// it, not silently as it arrives.
//
// Everything here is untrusted input in the fullest sense - hand-edited, from
// another vendor's tool, from another machine - so the line is parsed into a
// typed record and nothing more is assumed about it (§5.6, §14).
METHOD ImportConfigSetLine : BOOL
VAR_INPUT
    Line   : STRING(480);
    Commit : BOOL;
END_VAR
VAR
    info   : ST_ConfigSetInfo;
    record : ST_ConfigRecord;
END_VAR
ImportConfigSetLine := FALSE;
IF NOT _M_SetOpAllowed() THEN
    _importOpen := FALSE;
    RETURN;
END_IF
IF _setJson.M_ParseHeader(Line := Line, Info := info) THEN
    _importOpen := FALSE;
    info.Used := TRUE;
    info.RecordCount := 0;
    IF NOT _configStore.M_SaveBegin(Info := info) THEN
        RETURN;
    END_IF
    _importOpen := TRUE;
    ConfigPersist.LastSetName := info.SetName;
    ImportConfigSetLine := TRUE;
    RETURN;
END_IF
IF NOT _importOpen THEN
    RETURN;                                // a record before its header: refuse
END_IF
IF _setJson.M_ParseRecord(Line := Line, Record := record) THEN
    ImportConfigSetLine := _configStore.M_SaveRecord(Record := record);
    IF NOT ImportConfigSetLine THEN
        _configStore.M_SaveAbort();
        _importOpen := FALSE;
        RETURN;
    END_IF
ELSIF NOT Commit THEN
    // Neither a header nor a record, and not the closing call: the document is
    // not one this build understands. Abort rather than commit a partial set.
    _configStore.M_SaveAbort();
    _importOpen := FALSE;
    RETURN;
END_IF
IF Commit THEN
    ImportConfigSetLine := _configStore.M_SaveCommit();
    _importOpen := FALSE;
    IF ImportConfigSetLine THEN
        _M_MarkPersistPending();
    END_IF
END_IF
END_METHOD

// §3.8b - take part of a set line. A request carries at most 255 characters
// and an exported line may hold 480, so a longer line arrives as pieces:
// More = TRUE holds this piece and waits for the next; the first piece without
// More completes the line, which is then imported exactly like a whole one.
//
// Joined by FB_ConfigSetJson.M_Join, which measures first: a line that would
// exceed its width is refused and the import aborted - never truncated. (Not
// CONCAT/LEN: those stop at 255, which is the very limit being crossed.)
METHOD ImportConfigSetPiece : BOOL
VAR_INPUT
    Piece  : STRING(255);
    More   : BOOL;
    Commit : BOOL;
END_VAR
VAR
    line : STRING(480);
END_VAR
ImportConfigSetPiece := FALSE;
IF NOT _M_SetOpAllowed() THEN
    _importPart := '';
    RETURN;
END_IF
line := _importPart;
IF NOT _setJson.M_Join(Tail := Piece, Line := line) THEN
    _importPart := '';
    IF _importOpen THEN
        _configStore.M_SaveAbort();
        _importOpen := FALSE;
    END_IF
    RETURN;
END_IF
IF More THEN
    _importPart := line;
    ImportConfigSetPiece := TRUE;             // held, not yet imported
    RETURN;
END_IF
_importPart := '';
ImportConfigSetPiece := ImportConfigSetLine(Line := line, Commit := Commit);
END_METHOD

METHOD M_SequenceAskDecision
VAR_INPUT
    Req : ST_DecisionRequest;
END_VAR
_M_AskDecision(Req := Req);
END_METHOD

METHOD M_SequenceAwait : BOOL
VAR_INPUT
    Idx : INT;
    Label : STRING(120);
    Ok : BOOL;
END_VAR
M_SequenceAwait := _M_Await(Idx := Idx, Label := Label, Ok := Ok);
END_METHOD

METHOD M_SequenceClearDecision
IF Decision.Prompt <> '' THEN
    _M_LogDecision(EventKey := 'std.audit.decisionWithdrawn',
        SourcePath := Decision.SourcePath, Option := 0);
END_IF
_M_ClearDecisionState();
END_METHOD

METHOD M_SequenceComplete
IF _mode = E_Mode.CHANGEOVER THEN
    _M_HostEvent(Kind := E_HostEventKind.CHANGEOVER_DONE, PartUid := '',
        Subject := 'Model', Value := Model.ModelCode,
        Verdict := E_Verdict.NONE, ReasonCode := E_Reason.NONE);
END_IF
_M_Complete();
END_METHOD

METHOD M_SequenceCountGood
CountGood();
END_METHOD

METHOD M_SequenceEndOfCycle : BOOL
M_SequenceEndOfCycle := _M_EndOfCycle();
END_METHOD

METHOD M_SequenceFault
VAR_INPUT
    Reason : E_Reason;
    DescriptionKey : STRING(255);
END_VAR
_M_Fault(Reason, DescriptionKey);
END_METHOD

METHOD M_SequencePartProcessed : BOOL
VAR_INPUT
    Verdict : E_Verdict;
    Reason : E_Reason;
END_VAR
M_SequencePartProcessed :=
    _M_PartProcessed(Verdict := Verdict, Reason := Reason);
END_METHOD

METHOD M_SequencePartReceived : BOOL
M_SequencePartReceived := _M_PartReceived();
END_METHOD

METHOD M_SequencePartRecord : BOOL
VAR_INPUT
    RecordName : STRING(64);
    Value : LREAL;
    Minimum : LREAL;
    Maximum : LREAL;
    Target : LREAL;
    EngUnit : STRING(16);
END_VAR
M_SequencePartRecord := _M_PartRecord(RecordName := RecordName,
    Value := Value, Minimum := Minimum, Maximum := Maximum, Target := Target,
    EngUnit := EngUnit);
END_METHOD

METHOD M_SequencePartStarted
_M_PartStarted();
END_METHOD

// §6.8 register an attached chain (idempotent, bounded). Called from
// FB_SequenceBase.M_Attach, never by project code.
METHOD M_SequenceRegister : BOOL
VAR_INPUT
    Seq : I_Sequence;
END_VAR
VAR
    i : INT;
END_VAR
M_SequenceRegister := FALSE;
IF Seq = 0 THEN
    RETURN;
END_IF
FOR i := 1 TO _sequenceCount DO
    IF _sequences[i] = Seq THEN
        M_SequenceRegister := TRUE;        // already attached: Setup ran again
        RETURN;
    END_IF
END_FOR
IF _sequenceCount >= PL_Fraktal.MAX_SEQUENCES THEN
    RETURN;                                // bounded; refused, never silently dropped
END_IF
_sequenceCount := _sequenceCount + 1;
_sequences[_sequenceCount] := Seq;
M_SequenceRegister := TRUE;
END_METHOD

// §6.10 — reset every attached chain's shared transition result once per
// PLC cycle, before _M_Dispatch drives any step action. This is why a project
// never calls M_BeginScan itself, and why an SFC/LD/FBD chart needs no wiring
// to be safe against a stale ADVANCE (O1).
METHOD PROTECTED _M_BeginSequenceScan
VAR
    i : INT;
END_VAR
// §6.12 — close out the legs the previous scan's dispatch stopped recording. A step
// is live exactly while its action keeps calling M_Step, which is the same fact the
// chart draws, so nothing has to be deregistered when a leg finishes. Sweeping legs
// rather than rows makes this ~10 iterations however long the chain is.
FOR i := 0 TO PL_Fraktal.MAX_PARALLEL_BRANCHES DO
    IF (ActiveSteps[i].RowIdx > 0) AND NOT _branchTouched[i] THEN
        // The row keeps how long it ran: the HMI polls too slowly to have timed it.
        SequenceSteps[ActiveSteps[i].RowIdx].LastDuration := ActiveSteps[i].Elapsed;
        ActiveSteps[i].RowIdx := 0;
        ActiveSteps[i].TimedOut := FALSE;
    END_IF
    _branchTouched[i] := FALSE;
END_FOR
FOR i := 1 TO _sequenceCount DO
    IF _sequences[i] <> 0 THEN
        _sequences[i].M_BeginScan();
    END_IF
END_FOR
END_METHOD

// §6.8 - restart every attached chain. The base calls it where a chain can never
// resume (first scan, mode change, abort, abort in error). Whether a fresh run
// command or an operator reset RESTARTS the chain or lets it resume where an
// error stopped it is the project's policy (§6.9(d)), so a project that wants a
// restart there calls this one line from OnCommandStart / OnOperatorReset.
METHOD PROTECTED _M_RestartSequences
VAR
    i : INT;
END_VAR
FOR i := 1 TO _sequenceCount DO
    IF _sequences[i] <> 0 THEN
        _sequences[i].M_Restart();
    END_IF
END_FOR
// A decision belongs to the chain step that asked it; a restarted chain asks again.
Decision.Prompt := '';
DecisionAnswer := 0;
END_METHOD

// §3.14 - an aborted mode chain is abandoned, never resumed: restart every
// attached chain so the next command starts at N000 (§6.8).
METHOD PROTECTED OnAbort : DINT
OnAbort := SUPER^.OnAbort();
_M_RestartSequences();
END_METHOD

// §3.14 - error-state abort abandons the chain the same way (§6.8).
METHOD PROTECTED OnAbortInError : DINT
OnAbortInError := SUPER^.OnAbortInError();
_M_RestartSequences();
END_METHOD

// §6.9(e) — a step said something worth recording that is not a failure.
// Deliberately does NOT touch _exec: no fault is adopted, _M_Dispatch keeps
// running, and the chain follows its own recovery path. The ring entry is
// AUTO_RESET come+gone (§8.3(c)) so it can never block the next Start.
METHOD M_SequenceWarn : BOOL
VAR_INPUT
    Diag : ST_Diagnostic;
END_VAR
VAR
    d    : ST_Diagnostic;
    slot : INT;
END_VAR
d := Diag;
IF d.SourcePath = '' THEN
    d.SourcePath := _name;
END_IF
F_RationalizeDiagnostic(Diag := d);   // §8.8 owns a registered reason's level
IF (_seqIndex >= 1) AND (_seqIndex <= SequenceStepCount) THEN
    SequenceSteps[_seqIndex].WarningActive := TRUE;
    // A message about THIS Unit has nowhere to drill; one about a child keeps the
    // child's path, so the chart links to the module the message is about.
    IF d.SourcePath = _name THEN
        _M_SequenceAnnotate(RowIdx := _seqIndex, IsError := FALSE,
            Key := d.Description, SourcePath := '');
    ELSE
        _M_SequenceAnnotate(RowIdx := _seqIndex, IsError := FALSE,
            Key := d.Description, SourcePath := d.SourcePath);
    END_IF
END_IF
slot := AlarmLog.Raise(Reason := d.ReasonCode, Text := d.Description,
    Source := d.SourcePath, Severity := d.Severity, Category := d.Category,
    ResetClass := E_ResetClass.AUTO_RESET);
IF slot > 0 THEN
    AlarmLog.Gone(Slot := slot);       // an occurrence, not a standing condition
END_IF
M_SequenceWarn := TRUE;
END_METHOD

// §6.9 — a step raised a first-out itself. Stamp the flow-chart row with the
// error and its link before adopting the diagnostic, so the §3.13 chart can mark
// the step red and drill into the module that actually failed even when the step
// passed Awaits := 0. Adopting the diagnostic stops the chain: _M_FaultDiag puts
// the Unit in ERROR and _M_Dispatch no longer runs.
METHOD M_SequenceRaise : BOOL
VAR_INPUT
    Diag     : ST_Diagnostic;
    LinkPath : STRING(255);
END_VAR
M_SequenceRaise := FALSE;
IF (_seqIndex >= 1) AND (_seqIndex <= SequenceStepCount) THEN
    SequenceSteps[_seqIndex].ErrorActive := TRUE;
    _M_SequenceAnnotate(RowIdx := _seqIndex, IsError := TRUE,
        Key := Diag.Description, SourcePath := LinkPath);
END_IF
_M_FaultDiag(Diag := Diag);
M_SequenceRaise := TRUE;
END_METHOD

// §6.9 — the ERROR state ended: clear the flow-chart error marks and re-arm
// every attached chain so the step that raised the fault re-evaluates its
// command. A project writes nothing for this (§1.1 O1).
METHOD PROTECTED _M_ResumeSequencesAfterError
VAR
    i : INT;
END_VAR
FOR i := 1 TO SequenceStepCount DO
    SequenceSteps[i].ErrorActive := FALSE;
END_FOR
_M_SequenceAnnotationClear(RowIdx := 0, IsError := TRUE);
FOR i := 1 TO _sequenceCount DO
    IF _sequences[i] <> 0 THEN
        _sequences[i].M_ResumeAfterError();
    END_IF
END_FOR
END_METHOD

// I_SequenceHost (§6.7/§6.8) — step record for a separately-compiled chain.
METHOD M_SequenceSetStep
VAR_INPUT
    StepNo : INT;
    StepName : STRING(120);
    Awaits : I_Module;
    AwaitingLabel : STRING(120);
    TimeClass : E_TimeClass;
    ExpectedTime : TIME;
    Branch : INT;
END_VAR
// §6.12 — a step on a concurrent LEG publishes its own row and nothing else. The
// Unit's CurrentStep, the §6.9 stall walk and the §8.11.4 profiler are singular by
// definition; letting a leg write them would make the walk report whichever leg
// happened to run last. A leg is timed and guarded on its own row instead, so
// _M_SetStep keeps the signature every inline chain already calls (§1.1 O1).
IF Branch > 0 THEN
    _M_RecordSequenceStep(StepNo := StepNo, StepName := StepName, Awaits := Awaits,
        AwaitingLabel := AwaitingLabel, TimeClass := TimeClass, ExpectedTime := ExpectedTime,
        Branch := Branch);
    RETURN;
END_IF
_M_SetStep(StepNo := StepNo, StepName := StepName,
    Awaits := Awaits, AwaitingLabel := AwaitingLabel, TimeClass := TimeClass,
    ExpectedTime := ExpectedTime);
END_METHOD

METHOD M_SequenceStepGate : BOOL
VAR_INPUT
    Steppable : BOOL;
END_VAR
M_SequenceStepGate := _M_StepGate(Steppable := Steppable);
END_METHOD

// §3.4/§8.11 — accept a pending Stop BETWEEN cycles: the open profile fragment
// (just the wait step) is abandoned, not published as a production cycle.
METHOD M_SequenceStopNow
Profiler.CycleAbandon();
_stopReq := FALSE;
Execute := FALSE;
_M_Complete();
END_METHOD

// §3.4 — a chain polls this at its between-cycles wait step.
METHOD M_SequenceStopPending : BOOL
M_SequenceStopPending := _stopReq AND (_exec = E_ExecState.BUSY);
END_METHOD

METHOD M_SequenceTakeDecision : INT
M_SequenceTakeDecision := _M_TakeDecision();
END_METHOD

// §7.6.1a — single gated entry for a HELD manual action (hold-to-run). Same
// gates as ManualCommandTo: this Unit in MANUAL (§3.4) and MANUAL access
// (§7.7). Held := TRUE latches the request; FALSE releases it immediately.
//
// The release is explicit AND the latch expires, deliberately both: an explicit
// release stops the motion the moment the operator lets go, and the deadline
// stops it when no release ever arrives because the client vanished. Relying on
// either alone leaves one of those two cases moving.
//
// Hold-to-run over a transport is NON-SAFETY (no dead-man, TC3 §7.6): the
// enabling device is the safety-rated fact, derived below from the §9 facet and
// carried to the module, which weighs it itself.
METHOD ManualHeldTo : BOOL
VAR_INPUT
    TargetPath : STRING(255);
    Value      : DINT;
    Held       : BOOL;
END_VAR
VAR
    auditSlot : INT;
END_VAR
ManualHeldTo := FALSE;
IF NOT Held THEN
    // A release is always honoured, whatever the mode or access says now. The
    // operator letting go must never depend on a gate that may have changed
    // since they took hold of it.
    _heldActive := FALSE;
    _heldPath := '';
    _heldValue := 0;
    ManualHeldTo := TRUE;
    RETURN;
END_IF
IF _mode <> E_Mode.MANUAL THEN
    auditSlot := AlarmLog.Raise(Reason := E_Reason.NONE,
        Text := 'std.audit.manualCommandWrongMode', Source := TargetPath,
        Severity := E_Severity.LOW, Category := E_Category.SYSTEM,
        ResetClass := E_ResetClass.AUTO_RESET);
    IF auditSlot > 0 THEN AlarmLog.Gone(Slot := auditSlot); END_IF
    RETURN;
END_IF
IF NOT Access.PermitsLogged(Gate := E_GatedAction.MANUAL) THEN
    RETURN;                              // §7.7 denial already audited
END_IF
// Prove the target accepts it BEFORE latching, so a hold on a module that
// refuses never becomes a standing request nobody can see the source of.
IF NOT _M_RouteHeld(TargetPath := TargetPath, Value := Value) THEN
    RETURN;
END_IF
_heldPath := TargetPath;
_heldValue := Value;
_heldActive := TRUE;
_heldSinceMs := TIME_TO_DWORD(TIME());
ManualHeldTo := TRUE;
END_METHOD

// §7.6.1a — derive the enabling-device fact from THIS root's §9 safety facet and
// carry it to the owning module through the registered-child walk.
//
// F_ManualEnable is the single place the fact is derived, so grepping for it
// lists every path by which motion is authorised by an enabling device. Until
// now it had no production caller at all - the capability existed and nothing
// reached it.
METHOD PROTECTED _M_RouteHeld : BOOL
VAR_INPUT
    TargetPath : STRING(255);
    Value      : DINT;
END_VAR
VAR
    enable : ST_ManualEnableStatus;
END_VAR
enable := F_ManualEnable(Safety := Safety);
_M_RouteHeld := M_ApplyHeld(Scope := TargetPath, Value := Value,
    Enable := enable);
END_METHOD

// §3.13/§3.10.2 — raise the manifest revision ONCE the flow chart has stopped
// growing, rather than once per row discovered.
//
// The rows are the manifest's largest and most volatile contributor and they
// appear one at a time as the chain visits them, so a per-row bump turned one
// mode entry into one full-manifest refetch per step. This waits for the burst
// to settle and then charges for it once.
//
// The delay is bounded and small (PL_Fraktal.CHART_REV_SETTLE_MS): the chart
// appears fractionally later and COMPLETE, instead of promptly and then being
// refetched fourteen more times.
METHOD PRIVATE _M_ChartRevCyclic
VAR
    elapsed : DWORD;
END_VAR
IF NOT _chartDirty THEN
    RETURN;
END_IF
// Unsigned subtraction, so the monotonic counter wrapping cannot fabricate a
// settled chart (TC3 §8.11).
elapsed := TIME_TO_DWORD(TIME()) - _chartTouchedMs;
IF elapsed < PL_Fraktal.CHART_REV_SETTLE_MS THEN
    RETURN;                            // still growing: let the burst finish
END_IF
_chartDirty := FALSE;
ConfigRev := ConfigRev + 1;
END_METHOD

// §7.6.1a — re-assert the latched hold every scan, and drop it when the client
// stops refreshing. The module's own freshness timer stops the motion; this
// stops the ROOT from going on asking for it.
METHOD PRIVATE _M_HeldCyclic
VAR
    elapsed : DWORD;
END_VAR
IF NOT _heldActive THEN
    RETURN;
END_IF
// Leaving MANUAL, or losing the access that granted it, ends the hold at once.
IF _mode <> E_Mode.MANUAL THEN
    _heldActive := FALSE;
    RETURN;
END_IF
IF NOT Access.Permits(Gate := E_GatedAction.MANUAL) THEN
    _heldActive := FALSE;
    RETURN;
END_IF
// Unsigned subtraction, so the monotonic counter wrapping cannot fabricate an
// expired hold (TC3 §8.11).
elapsed := TIME_TO_DWORD(TIME()) - _heldSinceMs;
IF elapsed > PL_Fraktal.MANUAL_HELD_REFRESH_MS THEN
    _heldActive := FALSE;                // client went quiet: let go for it
    RETURN;
END_IF
_M_RouteHeld(TargetPath := _heldPath, Value := _heldValue);
END_METHOD

